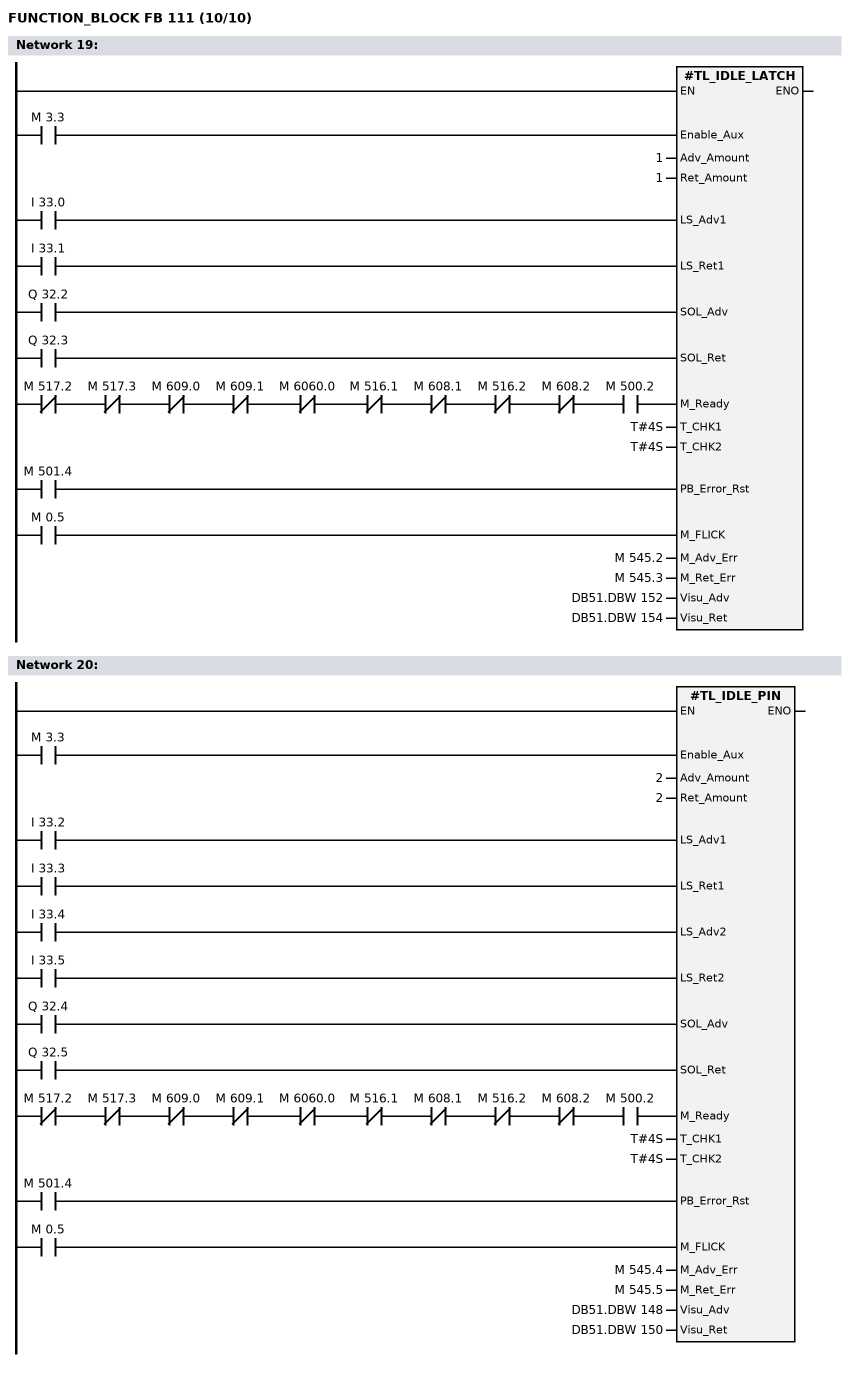

      A     M      3.3;
      =     L      0.0;
      BLD   103;
      A     I     33.0;
      =     L      0.1;
      BLD   103;
      A     I     33.1;
      =     L      0.2;
      BLD   103;
      A     Q     32.2;
      =     L      1.1;
      BLD   103;
      A     Q     32.3;
      =     L      1.2;
      BLD   103;
      AN    M    517.2;
      AN    M    517.3;
      AN    M    609.0;
      AN    M    609.1;
      AN    M   6060.0;
      AN    M    516.1;
      AN    M    608.1;
      AN    M    516.2;
      AN    M    608.2;
      A     M    500.2;
      =     L      1.3;
      BLD   103;
      A     M    501.4;
      =     L      1.5;
      BLD   103;
      A     M      0.5;
      =     L      1.6;
      BLD   103;
      CALL #TL_IDLE_LATCH (
           Enable_Aux               := L      0.0,
           Adv_Amount               := 1,
           Ret_Amount               := 1,
           LS_Adv1                  := L      0.1,
           LS_Ret1                  := L      0.2,
           SOL_Adv                  := L      1.1,
           SOL_Ret                  := L      1.2,
           M_Ready                  := L      1.3,
           T_CHK1                   := T#4S,
           T_CHK2                   := T#4S,
           PB_Error_Rst             := L      1.5,
           M_FLICK                  := L      1.6,
           M_Adv_Err                := M    545.2,
           M_Ret_Err                := M    545.3,
           Visu_Adv                 := DB51.DBW  152,
           Visu_Ret                 := DB51.DBW  154);
      NOP   0;
NETWORK
TITLE =

      A     M      3.3;
      =     L      0.0;
      BLD   103;
      A     I     33.2;
      =     L      0.1;
      BLD   103;
      A     I     33.3;
      =     L      0.2;
      BLD   103;
      A     I     33.4;
      =     L      0.3;
      BLD   103;
      A     I     33.5;
      =     L      0.4;
      BLD   103;
      A     Q     32.4;
      =     L      1.1;
      BLD   103;
      A     Q     32.5;
      =     L      1.2;
      BLD   103;
      AN    M    517.2;
      AN    M    517.3;
      AN    M    609.0;
      AN    M    609.1;
      AN    M   6060.0;
      AN    M    516.1;
      AN    M    608.1;
      AN    M    516.2;
      AN    M    608.2;
      A     M    500.2;
      =     L      1.3;
      BLD   103;
      A     M    501.4;
      =     L      1.5;
      BLD   103;
      A     M      0.5;
      =     L      1.6;
      BLD   103;
      CALL #TL_IDLE_PIN (
           Enable_Aux               := L      0.0,
           Adv_Amount               := 2,
           Ret_Amount               := 2,
           LS_Adv1                  := L      0.1,
           LS_Ret1                  := L      0.2,
           LS_Adv2                  := L      0.3,
           LS_Ret2                  := L      0.4,
           SOL_Adv                  := L      1.1,
           SOL_Ret                  := L      1.2,
           M_Ready                  := L      1.3,
           T_CHK1                   := T#4S,
           T_CHK2                   := T#4S,
           PB_Error_Rst             := L      1.5,
           M_FLICK                  := L      1.6,
           M_Adv_Err                := M    545.4,
           M_Ret_Err                := M    545.5,
           Visu_Adv                 := DB51.DBW  148,
           Visu_Ret                 := DB51.DBW  150);
      NOP   0;
END_FUNCTION_BLOCK

DATA_BLOCK DB 111
TITLE =
VERSION : 0.0

 FB 111
BEGIN
   LM_PIN.Enable_Aux := FALSE;
   LM_PIN.Adv_Amount := 0;
   LM_PIN.Ret_Amount := 0;
   LM_PIN.LS_Adv1 := FALSE;
   LM_PIN.LS_Ret1 := FALSE;
   LM_PIN.LS_Adv2 := FALSE;
   LM_PIN.LS_Ret2 := FALSE;
   LM_PIN.LS_Adv3 := FALSE;
   LM_PIN.LS_Ret3 := FALSE;
   LM_PIN.LS_Adv4 := FALSE;
   LM_PIN.LS_Ret4 := FALSE;
   LM_PIN.SOL_Adv := FALSE;
   LM_PIN.SOL_Ret := FALSE;
   LM_PIN.M_Ready := FALSE;
   LM_PIN.T_CHK1 := T#0MS;
   LM_PIN.T_CHK2 := T#0MS;
   LM_PIN.PB_Lamp_CHK := FALSE;
   LM_PIN.PB_Error_Rst := FALSE;
   LM_PIN.M_FLICK := FALSE;
   LM_PIN.M_Adv_Err := FALSE;
   LM_PIN.M_Ret_Err := FALSE;
   LM_PIN.LP_Adv := FALSE;
   LM_PIN.LP_Ret := FALSE;
   LM_PIN.Visu_Adv := W#16#0;
   LM_PIN.Visu_Ret := W#16#0;
   LM_PIN.Error_T1.IN := FALSE;
   LM_PIN.Error_T1.PT := T#0MS;
   LM_PIN.Error_T1.Q := FALSE;
   LM_PIN.Error_T1.ET := T#0MS;
   LM_PIN.Error_T1.STATE := B#16#0;
   LM_PIN.Error_T1.STIME := T#0MS;
   LM_PIN.Error_T1.ATIME := T#0MS;
   LM_PIN.Error_T2.IN := FALSE;
   LM_PIN.Error_T2.PT := T#0MS;
   LM_PIN.Error_T2.Q := FALSE;
   LM_PIN.Error_T2.ET := T#0MS;
   LM_PIN.Error_T2.STATE := B#16#0;
   LM_PIN.Error_T2.STIME := T#0MS;
   LM_PIN.Error_T2.ATIME := T#0MS;
   LM_PIN.CHK_Aux1 := FALSE;
   LM_PIN.CHK_Aux2 := FALSE;
   LM_PIN.Error_T1_DN := FALSE;
   LM_PIN.Error_T2_DN := FALSE;
   LM_PIN.Adv_Memo := FALSE;
   LM_PIN.Visu_Adv_Arr[0] := FALSE;
   LM_PIN.Visu_Adv_Arr[1] := FALSE;
   LM_PIN.Visu_Adv_Arr[2] := FALSE;
   LM_PIN.Visu_Adv_Arr[3] := FALSE;
   LM_PIN.Visu_Adv_Arr[4] := FALSE;
   LM_PIN.Visu_Adv_Arr[5] := FALSE;
   LM_PIN.Visu_Adv_Arr[6] := FALSE;
   LM_PIN.Visu_Adv_Arr[7] := FALSE;
   LM_PIN.Visu_Adv_Arr[8] := FALSE;
   LM_PIN.Visu_Adv_Arr[9] := FALSE;
   LM_PIN.Visu_Adv_Arr[10] := FALSE;
   LM_PIN.Visu_Adv_Arr[11] := FALSE;
   LM_PIN.Visu_Adv_Arr[12] := FALSE;
   LM_PIN.Visu_Adv_Arr[13] := FALSE;
   LM_PIN.Visu_Adv_Arr[14] := FALSE;
   LM_PIN.Visu_Adv_Arr[15] := FALSE;
   LM_PIN.Visu_Ret_Arr[0] := FALSE;
   LM_PIN.Visu_Ret_Arr[1] := FALSE;
   LM_PIN.Visu_Ret_Arr[2] := FALSE;
   LM_PIN.Visu_Ret_Arr[3] := FALSE;
   LM_PIN.Visu_Ret_Arr[4] := FALSE;
   LM_PIN.Visu_Ret_Arr[5] := FALSE;
   LM_PIN.Visu_Ret_Arr[6] := FALSE;
   LM_PIN.Visu_Ret_Arr[7] := FALSE;
   LM_PIN.Visu_Ret_Arr[8] := FALSE;
   LM_PIN.Visu_Ret_Arr[9] := FALSE;
   LM_PIN.Visu_Ret_Arr[10] := FALSE;
   LM_PIN.Visu_Ret_Arr[11] := FALSE;
   LM_PIN.Visu_Ret_Arr[12] := FALSE;
   LM_PIN.Visu_Ret_Arr[13] := FALSE;
   LM_PIN.Visu_Ret_Arr[14] := FALSE;
   LM_PIN.Visu_Ret_Arr[15] := FALSE;
   LM_PIN.BLK_Move_Ret := 0;
   LM_PIN.Enable := FALSE;
   LM_PIN.Adv_End := FALSE;
   LM_PIN.Ret_End := FALSE;
   LM_CLAMP1.Enable_Aux := FALSE;
   LM_CLAMP1.Adv_Amount := 0;
   LM_CLAMP1.Ret_Amount := 0;
   LM_CLAMP1.LS_Adv1 := FALSE;
   LM_CLAMP1.LS_Ret1 := FALSE;
   LM_CLAMP1.LS_Adv2 := FALSE;
   LM_CLAMP1.LS_Ret2 := FALSE;
   LM_CLAMP1.LS_Adv3 := FALSE;
   LM_CLAMP1.LS_Ret3 := FALSE;
   LM_CLAMP1.LS_Adv4 := FALSE;
   LM_CLAMP1.LS_Ret4 := FALSE;
   LM_CLAMP1.SOL_Adv := FALSE;
   LM_CLAMP1.SOL_Ret := FALSE;
   LM_CLAMP1.M_Ready := FALSE;
   LM_CLAMP1.T_CHK1 := T#0MS;
   LM_CLAMP1.T_CHK2 := T#0MS;
   LM_CLAMP1.PB_Lamp_CHK := FALSE;
   LM_CLAMP1.PB_Error_Rst := FALSE;
   LM_CLAMP1.M_FLICK := FALSE;
   LM_CLAMP1.M_Adv_Err := FALSE;
   LM_CLAMP1.M_Ret_Err := FALSE;
   LM_CLAMP1.LP_Adv := FALSE;
   LM_CLAMP1.LP_Ret := FALSE;
   LM_CLAMP1.Visu_Adv := W#16#0;
   LM_CLAMP1.Visu_Ret := W#16#0;
   LM_CLAMP1.Error_T1.IN := FALSE;
   LM_CLAMP1.Error_T1.PT := T#0MS;
   LM_CLAMP1.Error_T1.Q := FALSE;
   LM_CLAMP1.Error_T1.ET := T#0MS;
   LM_CLAMP1.Error_T1.STATE := B#16#0;
   LM_CLAMP1.Error_T1.STIME := T#0MS;
   LM_CLAMP1.Error_T1.ATIME := T#0MS;
   LM_CLAMP1.Error_T2.IN := FALSE;
   LM_CLAMP1.Error_T2.PT := T#0MS;
   LM_CLAMP1.Error_T2.Q := FALSE;
   LM_CLAMP1.Error_T2.ET := T#0MS;
   LM_CLAMP1.Error_T2.STATE := B#16#0;
   LM_CLAMP1.Error_T2.STIME := T#0MS;
   LM_CLAMP1.Error_T2.ATIME := T#0MS;
   LM_CLAMP1.CHK_Aux1 := FALSE;
   LM_CLAMP1.CHK_Aux2 := FALSE;
   LM_CLAMP1.Error_T1_DN := FALSE;
   LM_CLAMP1.Error_T2_DN := FALSE;
   LM_CLAMP1.Adv_Memo := FALSE;
   LM_CLAMP1.Visu_Adv_Arr[0] := FALSE;
   LM_CLAMP1.Visu_Adv_Arr[1] := FALSE;
   LM_CLAMP1.Visu_Adv_Arr[2] := FALSE;
   LM_CLAMP1.Visu_Adv_Arr[3] := FALSE;
   LM_CLAMP1.Visu_Adv_Arr[4] := FALSE;
   LM_CLAMP1.Visu_Adv_Arr[5] := FALSE;
   LM_CLAMP1.Visu_Adv_Arr[6] := FALSE;
   LM_CLAMP1.Visu_Adv_Arr[7] := FALSE;
   LM_CLAMP1.Visu_Adv_Arr[8] := FALSE;
   LM_CLAMP1.Visu_Adv_Arr[9] := FALSE;
   LM_CLAMP1.Visu_Adv_Arr[10] := FALSE;
   LM_CLAMP1.Visu_Adv_Arr[11] := FALSE;
   LM_CLAMP1.Visu_Adv_Arr[12] := FALSE;
   LM_CLAMP1.Visu_Adv_Arr[13] := FALSE;
   LM_CLAMP1.Visu_Adv_Arr[14] := FALSE;
   LM_CLAMP1.Visu_Adv_Arr[15] := FALSE;
   LM_CLAMP1.Visu_Ret_Arr[0] := FALSE;
   LM_CLAMP1.Visu_Ret_Arr[1] := FALSE;
   LM_CLAMP1.Visu_Ret_Arr[2] := FALSE;
   LM_CLAMP1.Visu_Ret_Arr[3] := FALSE;
   LM_CLAMP1.Visu_Ret_Arr[4] := FALSE;
   LM_CLAMP1.Visu_Ret_Arr[5] := FALSE;
   LM_CLAMP1.Visu_Ret_Arr[6] := FALSE;
   LM_CLAMP1.Visu_Ret_Arr[7] := FALSE;
   LM_CLAMP1.Visu_Ret_Arr[8] := FALSE;
   LM_CLAMP1.Visu_Ret_Arr[9] := FALSE;
   LM_CLAMP1.Visu_Ret_Arr[10] := FALSE;
   LM_CLAMP1.Visu_Ret_Arr[11] := FALSE;
   LM_CLAMP1.Visu_Ret_Arr[12] := FALSE;
   LM_CLAMP1.Visu_Ret_Arr[13] := FALSE;
   LM_CLAMP1.Visu_Ret_Arr[14] := FALSE;
   LM_CLAMP1.Visu_Ret_Arr[15] := FALSE;
   LM_CLAMP1.BLK_Move_Ret := 0;
   LM_CLAMP1.Enable := FALSE;
   LM_CLAMP1.Adv_End := FALSE;
   LM_CLAMP1.Ret_End := FALSE;
   LM_CLAMP2.Enable_Aux := FALSE;
   LM_CLAMP2.Adv_Amount := 0;
   LM_CLAMP2.Ret_Amount := 0;
   LM_CLAMP2.LS_Adv1 := FALSE;
   LM_CLAMP2.LS_Ret1 := FALSE;
   LM_CLAMP2.LS_Adv2 := FALSE;
   LM_CLAMP2.LS_Ret2 := FALSE;
   LM_CLAMP2.LS_Adv3 := FALSE;
   LM_CLAMP2.LS_Ret3 := FALSE;
   LM_CLAMP2.LS_Adv4 := FALSE;
   LM_CLAMP2.LS_Ret4 := FALSE;
   LM_CLAMP2.SOL_Adv := FALSE;
   LM_CLAMP2.SOL_Ret := FALSE;
   LM_CLAMP2.M_Ready := FALSE;
   LM_CLAMP2.T_CHK1 := T#0MS;
   LM_CLAMP2.T_CHK2 := T#0MS;
   LM_CLAMP2.PB_Lamp_CHK := FALSE;
   LM_CLAMP2.PB_Error_Rst := FALSE;
   LM_CLAMP2.M_FLICK := FALSE;
   LM_CLAMP2.M_Adv_Err := FALSE;
   LM_CLAMP2.M_Ret_Err := FALSE;
   LM_CLAMP2.LP_Adv := FALSE;
   LM_CLAMP2.LP_Ret := FALSE;
   LM_CLAMP2.Visu_Adv := W#16#0;
   LM_CLAMP2.Visu_Ret := W#16#0;
   LM_CLAMP2.Error_T1.IN := FALSE;
   LM_CLAMP2.Error_T1.PT := T#0MS;
   LM_CLAMP2.Error_T1.Q := FALSE;
   LM_CLAMP2.Error_T1.ET := T#0MS;
   LM_CLAMP2.Error_T1.STATE := B#16#0;
   LM_CLAMP2.Error_T1.STIME := T#0MS;
   LM_CLAMP2.Error_T1.ATIME := T#0MS;
   LM_CLAMP2.Error_T2.IN := FALSE;
   LM_CLAMP2.Error_T2.PT := T#0MS;
   LM_CLAMP2.Error_T2.Q := FALSE;
   LM_CLAMP2.Error_T2.ET := T#0MS;
   LM_CLAMP2.Error_T2.STATE := B#16#0;
   LM_CLAMP2.Error_T2.STIME := T#0MS;
   LM_CLAMP2.Error_T2.ATIME := T#0MS;
   LM_CLAMP2.CHK_Aux1 := FALSE;
   LM_CLAMP2.CHK_Aux2 := FALSE;
   LM_CLAMP2.Error_T1_DN := FALSE;
   LM_CLAMP2.Error_T2_DN := FALSE;
   LM_CLAMP2.Adv_Memo := FALSE;
   LM_CLAMP2.Visu_Adv_Arr[0] := FALSE;
   LM_CLAMP2.Visu_Adv_Arr[1] := FALSE;
   LM_CLAMP2.Visu_Adv_Arr[2] := FALSE;
   LM_CLAMP2.Visu_Adv_Arr[3] := FALSE;
   LM_CLAMP2.Visu_Adv_Arr[4] := FALSE;
   LM_CLAMP2.Visu_Adv_Arr[5] := FALSE;
   LM_CLAMP2.Visu_Adv_Arr[6] := FALSE;
   LM_CLAMP2.Visu_Adv_Arr[7] := FALSE;
   LM_CLAMP2.Visu_Adv_Arr[8] := FALSE;
   LM_CLAMP2.Visu_Adv_Arr[9] := FALSE;
   LM_CLAMP2.Visu_Adv_Arr[10] := FALSE;
   LM_CLAMP2.Visu_Adv_Arr[11] := FALSE;
   LM_CLAMP2.Visu_Adv_Arr[12] := FALSE;
   LM_CLAMP2.Visu_Adv_Arr[13] := FALSE;
   LM_CLAMP2.Visu_Adv_Arr[14] := FALSE;
   LM_CLAMP2.Visu_Adv_Arr[15] := FALSE;
   LM_CLAMP2.Visu_Ret_Arr[0] := FALSE;
   LM_CLAMP2.Visu_Ret_Arr[1] := FALSE;
   LM_CLAMP2.Visu_Ret_Arr[2] := FALSE;
   LM_CLAMP2.Visu_Ret_Arr[3] := FALSE;
   LM_CLAMP2.Visu_Ret_Arr[4] := FALSE;
   LM_CLAMP2.Visu_Ret_Arr[5] := FALSE;
   LM_CLAMP2.Visu_Ret_Arr[6] := FALSE;
   LM_CLAMP2.Visu_Ret_Arr[7] := FALSE;
   LM_CLAMP2.Visu_Ret_Arr[8] := FALSE;
   LM_CLAMP2.Visu_Ret_Arr[9] := FALSE;
   LM_CLAMP2.Visu_Ret_Arr[10] := FALSE;
   LM_CLAMP2.Visu_Ret_Arr[11] := FALSE;
   LM_CLAMP2.Visu_Ret_Arr[12] := FALSE;
   LM_CLAMP2.Visu_Ret_Arr[13] := FALSE;
   LM_CLAMP2.Visu_Ret_Arr[14] := FALSE;
   LM_CLAMP2.Visu_Ret_Arr[15] := FALSE;
   LM_CLAMP2.BLK_Move_Ret := 0;
   LM_CLAMP2.Enable := FALSE;
   LM_CLAMP2.Adv_End := FALSE;
   LM_CLAMP2.Ret_End := FALSE;
   LM_SLIDE.Enable_Aux := FALSE;
   LM_SLIDE.Adv_Amount := 0;
   LM_SLIDE.Ret_Amount := 0;
   LM_SLIDE.LS_Adv1 := FALSE;
   LM_SLIDE.LS_Ret1 := FALSE;
   LM_SLIDE.LS_Adv2 := FALSE;
   LM_SLIDE.LS_Ret2 := FALSE;
   LM_SLIDE.LS_Adv3 := FALSE;
   LM_SLIDE.LS_Ret3 := FALSE;
   LM_SLIDE.LS_Adv4 := FALSE;
   LM_SLIDE.LS_Ret4 := FALSE;
   LM_SLIDE.SOL_Adv := FALSE;
   LM_SLIDE.SOL_Ret := FALSE;
   LM_SLIDE.M_Ready := FALSE;
   LM_SLIDE.T_CHK1 := T#0MS;
   LM_SLIDE.T_CHK2 := T#0MS;
   LM_SLIDE.PB_Lamp_CHK := FALSE;
   LM_SLIDE.PB_Error_Rst := FALSE;
   LM_SLIDE.M_FLICK := FALSE;
   LM_SLIDE.M_Adv_Err := FALSE;
   LM_SLIDE.M_Ret_Err := FALSE;
   LM_SLIDE.LP_Adv := FALSE;
   LM_SLIDE.LP_Ret := FALSE;
   LM_SLIDE.Visu_Adv := W#16#0;
   LM_SLIDE.Visu_Ret := W#16#0;
   LM_SLIDE.Error_T1.IN := FALSE;
   LM_SLIDE.Error_T1.PT := T#0MS;
   LM_SLIDE.Error_T1.Q := FALSE;
   LM_SLIDE.Error_T1.ET := T#0MS;
   LM_SLIDE.Error_T1.STATE := B#16#0;
   LM_SLIDE.Error_T1.STIME := T#0MS;
   LM_SLIDE.Error_T1.ATIME := T#0MS;
   LM_SLIDE.Error_T2.IN := FALSE;
   LM_SLIDE.Error_T2.PT := T#0MS;
   LM_SLIDE.Error_T2.Q := FALSE;
   LM_SLIDE.Error_T2.ET := T#0MS;
   LM_SLIDE.Error_T2.STATE := B#16#0;
   LM_SLIDE.Error_T2.STIME := T#0MS;
   LM_SLIDE.Error_T2.ATIME := T#0MS;
   LM_SLIDE.CHK_Aux1 := FALSE;
   LM_SLIDE.CHK_Aux2 := FALSE;
   LM_SLIDE.Error_T1_DN := FALSE;
   LM_SLIDE.Error_T2_DN := FALSE;
   LM_SLIDE.Adv_Memo := FALSE;
   LM_SLIDE.Visu_Adv_Arr[0] := FALSE;
   LM_SLIDE.Visu_Adv_Arr[1] := FALSE;
   LM_SLIDE.Visu_Adv_Arr[2] := FALSE;
   LM_SLIDE.Visu_Adv_Arr[3] := FALSE;
   LM_SLIDE.Visu_Adv_Arr[4] := FALSE;
   LM_SLIDE.Visu_Adv_Arr[5] := FALSE;
   LM_SLIDE.Visu_Adv_Arr[6] := FALSE;
   LM_SLIDE.Visu_Adv_Arr[7] := FALSE;
   LM_SLIDE.Visu_Adv_Arr[8] := FALSE;
   LM_SLIDE.Visu_Adv_Arr[9] := FALSE;
   LM_SLIDE.Visu_Adv_Arr[10] := FALSE;
   LM_SLIDE.Visu_Adv_Arr[11] := FALSE;
   LM_SLIDE.Visu_Adv_Arr[12] := FALSE;
   LM_SLIDE.Visu_Adv_Arr[13] := FALSE;
   LM_SLIDE.Visu_Adv_Arr[14] := FALSE;
   LM_SLIDE.Visu_Adv_Arr[15] := FALSE;
   LM_SLIDE.Visu_Ret_Arr[0] := FALSE;
   LM_SLIDE.Visu_Ret_Arr[1] := FALSE;
   LM_SLIDE.Visu_Ret_Arr[2] := FALSE;
   LM_SLIDE.Visu_Ret_Arr[3] := FALSE;
   LM_SLIDE.Visu_Ret_Arr[4] := FALSE;
   LM_SLIDE.Visu_Ret_Arr[5] := FALSE;
   LM_SLIDE.Visu_Ret_Arr[6] := FALSE;
   LM_SLIDE.Visu_Ret_Arr[7] := FALSE;
   LM_SLIDE.Visu_Ret_Arr[8] := FALSE;
   LM_SLIDE.Visu_Ret_Arr[9] := FALSE;
   LM_SLIDE.Visu_Ret_Arr[10] := FALSE;
   LM_SLIDE.Visu_Ret_Arr[11] := FALSE;
   LM_SLIDE.Visu_Ret_Arr[12] := FALSE;
   LM_SLIDE.Visu_Ret_Arr[13] := FALSE;
   LM_SLIDE.Visu_Ret_Arr[14] := FALSE;
   LM_SLIDE.Visu_Ret_Arr[15] := FALSE;
   LM_SLIDE.BLK_Move_Ret := 0;
   LM_SLIDE.Enable := FALSE;
   LM_SLIDE.Adv_End := FALSE;
   LM_SLIDE.Ret_End := FALSE;
   LM_SLIDE_ADV_LOCK.Enable_Aux := FALSE;
   LM_SLIDE_ADV_LOCK.Adv_Amount := 0;
   LM_SLIDE_ADV_LOCK.Ret_Amount := 0;
   LM_SLIDE_ADV_LOCK.LS_Adv1 := FALSE;
   LM_SLIDE_ADV_LOCK.LS_Ret1 := FALSE;
   LM_SLIDE_ADV_LOCK.LS_Adv2 := FALSE;
   LM_SLIDE_ADV_LOCK.LS_Ret2 := FALSE;
   LM_SLIDE_ADV_LOCK.LS_Adv3 := FALSE;
   LM_SLIDE_ADV_LOCK.LS_Ret3 := FALSE;
   LM_SLIDE_ADV_LOCK.LS_Adv4 := FALSE;
   LM_SLIDE_ADV_LOCK.LS_Ret4 := FALSE;
   LM_SLIDE_ADV_LOCK.SOL_Adv := FALSE;
   LM_SLIDE_ADV_LOCK.SOL_Ret := FALSE;
   LM_SLIDE_ADV_LOCK.M_Ready := FALSE;
   LM_SLIDE_ADV_LOCK.T_CHK1 := T#0MS;
   LM_SLIDE_ADV_LOCK.T_CHK2 := T#0MS;
   LM_SLIDE_ADV_LOCK.PB_Lamp_CHK := FALSE;
   LM_SLIDE_ADV_LOCK.PB_Error_Rst := FALSE;
   LM_SLIDE_ADV_LOCK.M_FLICK := FALSE;
   LM_SLIDE_ADV_LOCK.M_Adv_Err := FALSE;
   LM_SLIDE_ADV_LOCK.M_Ret_Err := FALSE;
   LM_SLIDE_ADV_LOCK.LP_Adv := FALSE;
   LM_SLIDE_ADV_LOCK.LP_Ret := FALSE;
   LM_SLIDE_ADV_LOCK.Visu_Adv := W#16#0;
   LM_SLIDE_ADV_LOCK.Visu_Ret := W#16#0;
   LM_SLIDE_ADV_LOCK.Error_T1.IN := FALSE;
   LM_SLIDE_ADV_LOCK.Error_T1.PT := T#0MS;
   LM_SLIDE_ADV_LOCK.Error_T1.Q := FALSE;
   LM_SLIDE_ADV_LOCK.Error_T1.ET := T#0MS;
   LM_SLIDE_ADV_LOCK.Error_T1.STATE := B#16#0;
   LM_SLIDE_ADV_LOCK.Error_T1.STIME := T#0MS;
   LM_SLIDE_ADV_LOCK.Error_T1.ATIME := T#0MS;
   LM_SLIDE_ADV_LOCK.Error_T2.IN := FALSE;
   LM_SLIDE_ADV_LOCK.Error_T2.PT := T#0MS;
   LM_SLIDE_ADV_LOCK.Error_T2.Q := FALSE;
   LM_SLIDE_ADV_LOCK.Error_T2.ET := T#0MS;
   LM_SLIDE_ADV_LOCK.Error_T2.STATE := B#16#0;
   LM_SLIDE_ADV_LOCK.Error_T2.STIME := T#0MS;
   LM_SLIDE_ADV_LOCK.Error_T2.ATIME := T#0MS;
   LM_SLIDE_ADV_LOCK.CHK_Aux1 := FALSE;
   LM_SLIDE_ADV_LOCK.CHK_Aux2 := FALSE;
   LM_SLIDE_ADV_LOCK.Error_T1_DN := FALSE;
   LM_SLIDE_ADV_LOCK.Error_T2_DN := FALSE;
   LM_SLIDE_ADV_LOCK.Adv_Memo := FALSE;
   LM_SLIDE_ADV_LOCK.Visu_Adv_Arr[0] := FALSE;
   LM_SLIDE_ADV_LOCK.Visu_Adv_Arr[1] := FALSE;
   LM_SLIDE_ADV_LOCK.Visu_Adv_Arr[2] := FALSE;
   LM_SLIDE_ADV_LOCK.Visu_Adv_Arr[3] := FALSE;
   LM_SLIDE_ADV_LOCK.Visu_Adv_Arr[4] := FALSE;
   LM_SLIDE_ADV_LOCK.Visu_Adv_Arr[5] := FALSE;
   LM_SLIDE_ADV_LOCK.Visu_Adv_Arr[6] := FALSE;
   LM_SLIDE_ADV_LOCK.Visu_Adv_Arr[7] := FALSE;
   LM_SLIDE_ADV_LOCK.Visu_Adv_Arr[8] := FALSE;
   LM_SLIDE_ADV_LOCK.Visu_Adv_Arr[9] := FALSE;
   LM_SLIDE_ADV_LOCK.Visu_Adv_Arr[10] := FALSE;
   LM_SLIDE_ADV_LOCK.Visu_Adv_Arr[11] := FALSE;
   LM_SLIDE_ADV_LOCK.Visu_Adv_Arr[12] := FALSE;
   LM_SLIDE_ADV_LOCK.Visu_Adv_Arr[13] := FALSE;
   LM_SLIDE_ADV_LOCK.Visu_Adv_Arr[14] := FALSE;
   LM_SLIDE_ADV_LOCK.Visu_Adv_Arr[15] := FALSE;
   LM_SLIDE_ADV_LOCK.Visu_Ret_Arr[0] := FALSE;
   LM_SLIDE_ADV_LOCK.Visu_Ret_Arr[1] := FALSE;
   LM_SLIDE_ADV_LOCK.Visu_Ret_Arr[2] := FALSE;
   LM_SLIDE_ADV_LOCK.Visu_Ret_Arr[3] := FALSE;
   LM_SLIDE_ADV_LOCK.Visu_Ret_Arr[4] := FALSE;
   LM_SLIDE_ADV_LOCK.Visu_Ret_Arr[5] := FALSE;
   LM_SLIDE_ADV_LOCK.Visu_Ret_Arr[6] := FALSE;
   LM_SLIDE_ADV_LOCK.Visu_Ret_Arr[7] := FALSE;
   LM_SLIDE_ADV_LOCK.Visu_Ret_Arr[8] := FALSE;
   LM_SLIDE_ADV_LOCK.Visu_Ret_Arr[9] := FALSE;
   LM_SLIDE_ADV_LOCK.Visu_Ret_Arr[10] := FALSE;
   LM_SLIDE_ADV_LOCK.Visu_Ret_Arr[11] := FALSE;
   LM_SLIDE_ADV_LOCK.Visu_Ret_Arr[12] := FALSE;
   LM_SLIDE_ADV_LOCK.Visu_Ret_Arr[13] := FALSE;
   LM_SLIDE_ADV_LOCK.Visu_Ret_Arr[14] := FALSE;
   LM_SLIDE_ADV_LOCK.Visu_Ret_Arr[15] := FALSE;
   LM_SLIDE_ADV_LOCK.BLK_Move_Ret := 0;
   LM_SLIDE_ADV_LOCK.Enable := FALSE;
   LM_SLIDE_ADV_LOCK.Adv_End := FALSE;
   LM_SLIDE_ADV_LOCK.Ret_End := FALSE;
   LM_GUN1_SHIFT.Enable_Aux := FALSE;
   LM_GUN1_SHIFT.Adv_Amount := 0;
   LM_GUN1_SHIFT.Ret_Amount := 0;
   LM_GUN1_SHIFT.LS_Adv1 := FALSE;
   LM_GUN1_SHIFT.LS_Ret1 := FALSE;
   LM_GUN1_SHIFT.LS_Adv2 := FALSE;
   LM_GUN1_SHIFT.LS_Ret2 := FALSE;
   LM_GUN1_SHIFT.LS_Adv3 := FALSE;
   LM_GUN1_SHIFT.LS_Ret3 := FALSE;
   LM_GUN1_SHIFT.LS_Adv4 := FALSE;
   LM_GUN1_SHIFT.LS_Ret4 := FALSE;
   LM_GUN1_SHIFT.SOL_Adv := FALSE;
   LM_GUN1_SHIFT.SOL_Ret := FALSE;
   LM_GUN1_SHIFT.M_Ready := FALSE;
   LM_GUN1_SHIFT.T_CHK1 := T#0MS;
   LM_GUN1_SHIFT.T_CHK2 := T#0MS;
   LM_GUN1_SHIFT.PB_Lamp_CHK := FALSE;
   LM_GUN1_SHIFT.PB_Error_Rst := FALSE;
   LM_GUN1_SHIFT.M_FLICK := FALSE;
   LM_GUN1_SHIFT.M_Adv_Err := FALSE;
   LM_GUN1_SHIFT.M_Ret_Err := FALSE;
   LM_GUN1_SHIFT.LP_Adv := FALSE;
   LM_GUN1_SHIFT.LP_Ret := FALSE;
   LM_GUN1_SHIFT.Visu_Adv := W#16#0;
   LM_GUN1_SHIFT.Visu_Ret := W#16#0;
   LM_GUN1_SHIFT.Error_T1.IN := FALSE;
   LM_GUN1_SHIFT.Error_T1.PT := T#0MS;
   LM_GUN1_SHIFT.Error_T1.Q := FALSE;
   LM_GUN1_SHIFT.Error_T1.ET := T#0MS;
   LM_GUN1_SHIFT.Error_T1.STATE := B#16#0;
   LM_GUN1_SHIFT.Error_T1.STIME := T#0MS;
   LM_GUN1_SHIFT.Error_T1.ATIME := T#0MS;
   LM_GUN1_SHIFT.Error_T2.IN := FALSE;
   LM_GUN1_SHIFT.Error_T2.PT := T#0MS;
   LM_GUN1_SHIFT.Error_T2.Q := FALSE;
   LM_GUN1_SHIFT.Error_T2.ET := T#0MS;
   LM_GUN1_SHIFT.Error_T2.STATE := B#16#0;
   LM_GUN1_SHIFT.Error_T2.STIME := T#0MS;
   LM_GUN1_SHIFT.Error_T2.ATIME := T#0MS;
   LM_GUN1_SHIFT.CHK_Aux1 := FALSE;
   LM_GUN1_SHIFT.CHK_Aux2 := FALSE;
   LM_GUN1_SHIFT.Error_T1_DN := FALSE;
   LM_GUN1_SHIFT.Error_T2_DN := FALSE;
   LM_GUN1_SHIFT.Adv_Memo := FALSE;
   LM_GUN1_SHIFT.Visu_Adv_Arr[0] := FALSE;
   LM_GUN1_SHIFT.Visu_Adv_Arr[1] := FALSE;
   LM_GUN1_SHIFT.Visu_Adv_Arr[2] := FALSE;
   LM_GUN1_SHIFT.Visu_Adv_Arr[3] := FALSE;
   LM_GUN1_SHIFT.Visu_Adv_Arr[4] := FALSE;
   LM_GUN1_SHIFT.Visu_Adv_Arr[5] := FALSE;
   LM_GUN1_SHIFT.Visu_Adv_Arr[6] := FALSE;
   LM_GUN1_SHIFT.Visu_Adv_Arr[7] := FALSE;
   LM_GUN1_SHIFT.Visu_Adv_Arr[8] := FALSE;
   LM_GUN1_SHIFT.Visu_Adv_Arr[9] := FALSE;
   LM_GUN1_SHIFT.Visu_Adv_Arr[10] := FALSE;
   LM_GUN1_SHIFT.Visu_Adv_Arr[11] := FALSE;
   LM_GUN1_SHIFT.Visu_Adv_Arr[12] := FALSE;
   LM_GUN1_SHIFT.Visu_Adv_Arr[13] := FALSE;
   LM_GUN1_SHIFT.Visu_Adv_Arr[14] := FALSE;
   LM_GUN1_SHIFT.Visu_Adv_Arr[15] := FALSE;
   LM_GUN1_SHIFT.Visu_Ret_Arr[0] := FALSE;
   LM_GUN1_SHIFT.Visu_Ret_Arr[1] := FALSE;
   LM_GUN1_SHIFT.Visu_Ret_Arr[2] := FALSE;
   LM_GUN1_SHIFT.Visu_Ret_Arr[3] := FALSE;
   LM_GUN1_SHIFT.Visu_Ret_Arr[4] := FALSE;
   LM_GUN1_SHIFT.Visu_Ret_Arr[5] := FALSE;
   LM_GUN1_SHIFT.Visu_Ret_Arr[6] := FALSE;
   LM_GUN1_SHIFT.Visu_Ret_Arr[7] := FALSE;
   LM_GUN1_SHIFT.Visu_Ret_Arr[8] := FALSE;
   LM_GUN1_SHIFT.Visu_Ret_Arr[9] := FALSE;
   LM_GUN1_SHIFT.Visu_Ret_Arr[10] := FALSE;
   LM_GUN1_SHIFT.Visu_Ret_Arr[11] := FALSE;
   LM_GUN1_SHIFT.Visu_Ret_Arr[12] := FALSE;
   LM_GUN1_SHIFT.Visu_Ret_Arr[13] := FALSE;
   LM_GUN1_SHIFT.Visu_Ret_Arr[14] := FALSE;
   LM_GUN1_SHIFT.Visu_Ret_Arr[15] := FALSE;
   LM_GUN1_SHIFT.BLK_Move_Ret := 0;
   LM_GUN1_SHIFT.Enable := FALSE;
   LM_GUN1_SHIFT.Adv_End := FALSE;
   LM_GUN1_SHIFT.Ret_End := FALSE;
   LM_GUN2_SHIFT.Enable_Aux := FALSE;
   LM_GUN2_SHIFT.Adv_Amount := 0;
   LM_GUN2_SHIFT.Ret_Amount := 0;
   LM_GUN2_SHIFT.LS_Adv1 := FALSE;
   LM_GUN2_SHIFT.LS_Ret1 := FALSE;
   LM_GUN2_SHIFT.LS_Adv2 := FALSE;
   LM_GUN2_SHIFT.LS_Ret2 := FALSE;
   LM_GUN2_SHIFT.LS_Adv3 := FALSE;
   LM_GUN2_SHIFT.LS_Ret3 := FALSE;
   LM_GUN2_SHIFT.LS_Adv4 := FALSE;
   LM_GUN2_SHIFT.LS_Ret4 := FALSE;
   LM_GUN2_SHIFT.SOL_Adv := FALSE;
   LM_GUN2_SHIFT.SOL_Ret := FALSE;
   LM_GUN2_SHIFT.M_Ready := FALSE;
   LM_GUN2_SHIFT.T_CHK1 := T#0MS;
   LM_GUN2_SHIFT.T_CHK2 := T#0MS;
   LM_GUN2_SHIFT.PB_Lamp_CHK := FALSE;
   LM_GUN2_SHIFT.PB_Error_Rst := FALSE;
   LM_GUN2_SHIFT.M_FLICK := FALSE;
   LM_GUN2_SHIFT.M_Adv_Err := FALSE;
   LM_GUN2_SHIFT.M_Ret_Err := FALSE;
   LM_GUN2_SHIFT.LP_Adv := FALSE;
   LM_GUN2_SHIFT.LP_Ret := FALSE;
   LM_GUN2_SHIFT.Visu_Adv := W#16#0;
   LM_GUN2_SHIFT.Visu_Ret := W#16#0;
   LM_GUN2_SHIFT.Error_T1.IN := FALSE;
   LM_GUN2_SHIFT.Error_T1.PT := T#0MS;
   LM_GUN2_SHIFT.Error_T1.Q := FALSE;
   LM_GUN2_SHIFT.Error_T1.ET := T#0MS;
   LM_GUN2_SHIFT.Error_T1.STATE := B#16#0;
   LM_GUN2_SHIFT.Error_T1.STIME := T#0MS;
   LM_GUN2_SHIFT.Error_T1.ATIME := T#0MS;
   LM_GUN2_SHIFT.Error_T2.IN := FALSE;
   LM_GUN2_SHIFT.Error_T2.PT := T#0MS;
   LM_GUN2_SHIFT.Error_T2.Q := FALSE;
   LM_GUN2_SHIFT.Error_T2.ET := T#0MS;
   LM_GUN2_SHIFT.Error_T2.STATE := B#16#0;
   LM_GUN2_SHIFT.Error_T2.STIME := T#0MS;
   LM_GUN2_SHIFT.Error_T2.ATIME := T#0MS;
   LM_GUN2_SHIFT.CHK_Aux1 := FALSE;
   LM_GUN2_SHIFT.CHK_Aux2 := FALSE;
   LM_GUN2_SHIFT.Error_T1_DN := FALSE;
   LM_GUN2_SHIFT.Error_T2_DN := FALSE;
   LM_GUN2_SHIFT.Adv_Memo := FALSE;
   LM_GUN2_SHIFT.Visu_Adv_Arr[0] := FALSE;
   LM_GUN2_SHIFT.Visu_Adv_Arr[1] := FALSE;
   LM_GUN2_SHIFT.Visu_Adv_Arr[2] := FALSE;
   LM_GUN2_SHIFT.Visu_Adv_Arr[3] := FALSE;
   LM_GUN2_SHIFT.Visu_Adv_Arr[4] := FALSE;
   LM_GUN2_SHIFT.Visu_Adv_Arr[5] := FALSE;
   LM_GUN2_SHIFT.Visu_Adv_Arr[6] := FALSE;
   LM_GUN2_SHIFT.Visu_Adv_Arr[7] := FALSE;
   LM_GUN2_SHIFT.Visu_Adv_Arr[8] := FALSE;
   LM_GUN2_SHIFT.Visu_Adv_Arr[9] := FALSE;
   LM_GUN2_SHIFT.Visu_Adv_Arr[10] := FALSE;
   LM_GUN2_SHIFT.Visu_Adv_Arr[11] := FALSE;
   LM_GUN2_SHIFT.Visu_Adv_Arr[12] := FALSE;
   LM_GUN2_SHIFT.Visu_Adv_Arr[13] := FALSE;
   LM_GUN2_SHIFT.Visu_Adv_Arr[14] := FALSE;
   LM_GUN2_SHIFT.Visu_Adv_Arr[15] := FALSE;
   LM_GUN2_SHIFT.Visu_Ret_Arr[0] := FALSE;
   LM_GUN2_SHIFT.Visu_Ret_Arr[1] := FALSE;
   LM_GUN2_SHIFT.Visu_Ret_Arr[2] := FALSE;
   LM_GUN2_SHIFT.Visu_Ret_Arr[3] := FALSE;
   LM_GUN2_SHIFT.Visu_Ret_Arr[4] := FALSE;
   LM_GUN2_SHIFT.Visu_Ret_Arr[5] := FALSE;
   LM_GUN2_SHIFT.Visu_Ret_Arr[6] := FALSE;
   LM_GUN2_SHIFT.Visu_Ret_Arr[7] := FALSE;
   LM_GUN2_SHIFT.Visu_Ret_Arr[8] := FALSE;
   LM_GUN2_SHIFT.Visu_Ret_Arr[9] := FALSE;
   LM_GUN2_SHIFT.Visu_Ret_Arr[10] := FALSE;
   LM_GUN2_SHIFT.Visu_Ret_Arr[11] := FALSE;
   LM_GUN2_SHIFT.Visu_Ret_Arr[12] := FALSE;
   LM_GUN2_SHIFT.Visu_Ret_Arr[13] := FALSE;
   LM_GUN2_SHIFT.Visu_Ret_Arr[14] := FALSE;
   LM_GUN2_SHIFT.Visu_Ret_Arr[15] := FALSE;
   LM_GUN2_SHIFT.BLK_Move_Ret := 0;
   LM_GUN2_SHIFT.Enable := FALSE;
   LM_GUN2_SHIFT.Adv_End := FALSE;
   LM_GUN2_SHIFT.Ret_End := FALSE;
   LM_GUN2_LATCH.Enable_Aux := FALSE;
   LM_GUN2_LATCH.Adv_Amount := 0;
   LM_GUN2_LATCH.Ret_Amount := 0;
   LM_GUN2_LATCH.LS_Adv1 := FALSE;
   LM_GUN2_LATCH.LS_Ret1 := FALSE;
   LM_GUN2_LATCH.LS_Adv2 := FALSE;
   LM_GUN2_LATCH.LS_Ret2 := FALSE;
   LM_GUN2_LATCH.LS_Adv3 := FALSE;
   LM_GUN2_LATCH.LS_Ret3 := FALSE;
   LM_GUN2_LATCH.LS_Adv4 := FALSE;
   LM_GUN2_LATCH.LS_Ret4 := FALSE;
   LM_GUN2_LATCH.SOL_Adv := FALSE;
   LM_GUN2_LATCH.SOL_Ret := FALSE;
   LM_GUN2_LATCH.M_Ready := FALSE;
   LM_GUN2_LATCH.T_CHK1 := T#0MS;
   LM_GUN2_LATCH.T_CHK2 := T#0MS;
   LM_GUN2_LATCH.PB_Lamp_CHK := FALSE;
   LM_GUN2_LATCH.PB_Error_Rst := FALSE;
   LM_GUN2_LATCH.M_FLICK := FALSE;
   LM_GUN2_LATCH.M_Adv_Err := FALSE;
   LM_GUN2_LATCH.M_Ret_Err := FALSE;
   LM_GUN2_LATCH.LP_Adv := FALSE;
   LM_GUN2_LATCH.LP_Ret := FALSE;
   LM_GUN2_LATCH.Visu_Adv := W#16#0;
   LM_GUN2_LATCH.Visu_Ret := W#16#0;
   LM_GUN2_LATCH.Error_T1.IN := FALSE;
   LM_GUN2_LATCH.Error_T1.PT := T#0MS;
   LM_GUN2_LATCH.Error_T1.Q := FALSE;
   LM_GUN2_LATCH.Error_T1.ET := T#0MS;
   LM_GUN2_LATCH.Error_T1.STATE := B#16#0;
   LM_GUN2_LATCH.Error_T1.STIME := T#0MS;
   LM_GUN2_LATCH.Error_T1.ATIME := T#0MS;
   LM_GUN2_LATCH.Error_T2.IN := FALSE;
   LM_GUN2_LATCH.Error_T2.PT := T#0MS;
   LM_GUN2_LATCH.Error_T2.Q := FALSE;
   LM_GUN2_LATCH.Error_T2.ET := T#0MS;
   LM_GUN2_LATCH.Error_T2.STATE := B#16#0;
   LM_GUN2_LATCH.Error_T2.STIME := T#0MS;
   LM_GUN2_LATCH.Error_T2.ATIME := T#0MS;
   LM_GUN2_LATCH.CHK_Aux1 := FALSE;
   LM_GUN2_LATCH.CHK_Aux2 := FALSE;
   LM_GUN2_LATCH.Error_T1_DN := FALSE;
   LM_GUN2_LATCH.Error_T2_DN := FALSE;
   LM_GUN2_LATCH.Adv_Memo := FALSE;
   LM_GUN2_LATCH.Visu_Adv_Arr[0] := FALSE;
   LM_GUN2_LATCH.Visu_Adv_Arr[1] := FALSE;
   LM_GUN2_LATCH.Visu_Adv_Arr[2] := FALSE;
   LM_GUN2_LATCH.Visu_Adv_Arr[3] := FALSE;
   LM_GUN2_LATCH.Visu_Adv_Arr[4] := FALSE;
   LM_GUN2_LATCH.Visu_Adv_Arr[5] := FALSE;
   LM_GUN2_LATCH.Visu_Adv_Arr[6] := FALSE;
   LM_GUN2_LATCH.Visu_Adv_Arr[7] := FALSE;
   LM_GUN2_LATCH.Visu_Adv_Arr[8] := FALSE;
   LM_GUN2_LATCH.Visu_Adv_Arr[9] := FALSE;
   LM_GUN2_LATCH.Visu_Adv_Arr[10] := FALSE;
   LM_GUN2_LATCH.Visu_Adv_Arr[11] := FALSE;
   LM_GUN2_LATCH.Visu_Adv_Arr[12] := FALSE;
   LM_GUN2_LATCH.Visu_Adv_Arr[13] := FALSE;
   LM_GUN2_LATCH.Visu_Adv_Arr[14] := FALSE;
   LM_GUN2_LATCH.Visu_Adv_Arr[15] := FALSE;
   LM_GUN2_LATCH.Visu_Ret_Arr[0] := FALSE;
   LM_GUN2_LATCH.Visu_Ret_Arr[1] := FALSE;
   LM_GUN2_LATCH.Visu_Ret_Arr[2] := FALSE;
   LM_GUN2_LATCH.Visu_Ret_Arr[3] := FALSE;
   LM_GUN2_LATCH.Visu_Ret_Arr[4] := FALSE;
   LM_GUN2_LATCH.Visu_Ret_Arr[5] := FALSE;
   LM_GUN2_LATCH.Visu_Ret_Arr[6] := FALSE;
   LM_GUN2_LATCH.Visu_Ret_Arr[7] := FALSE;
   LM_GUN2_LATCH.Visu_Ret_Arr[8] := FALSE;
   LM_GUN2_LATCH.Visu_Ret_Arr[9] := FALSE;
   LM_GUN2_LATCH.Visu_Ret_Arr[10] := FALSE;
   LM_GUN2_LATCH.Visu_Ret_Arr[11] := FALSE;
   LM_GUN2_LATCH.Visu_Ret_Arr[12] := FALSE;
   LM_GUN2_LATCH.Visu_Ret_Arr[13] := FALSE;
   LM_GUN2_LATCH.Visu_Ret_Arr[14] := FALSE;
   LM_GUN2_LATCH.Visu_Ret_Arr[15] := FALSE;
   LM_GUN2_LATCH.BLK_Move_Ret := 0;
   LM_GUN2_LATCH.Enable := FALSE;
   LM_GUN2_LATCH.Adv_End := FALSE;
   LM_GUN2_LATCH.Ret_End := FALSE;
   TL_SLIDE.Enable_Aux := FALSE;
   TL_SLIDE.Adv_Amount := 0;
   TL_SLIDE.Ret_Amount := 0;
   TL_SLIDE.LS_Adv1 := FALSE;
   TL_SLIDE.LS_Ret1 := FALSE;
   TL_SLIDE.LS_Adv2 := FALSE;
   TL_SLIDE.LS_Ret2 := FALSE;
   TL_SLIDE.LS_Adv3 := FALSE;
   TL_SLIDE.LS_Ret3 := FALSE;
   TL_SLIDE.LS_Adv4 := FALSE;
   TL_SLIDE.LS_Ret4 := FALSE;
   TL_SLIDE.SOL_Adv := FALSE;
   TL_SLIDE.SOL_Ret := FALSE;
   TL_SLIDE.M_Ready := FALSE;
   TL_SLIDE.T_CHK1 := T#0MS;
   TL_SLIDE.T_CHK2 := T#0MS;
   TL_SLIDE.PB_Lamp_CHK := FALSE;
   TL_SLIDE.PB_Error_Rst := FALSE;
   TL_SLIDE.M_FLICK := FALSE;
   TL_SLIDE.M_Adv_Err := FALSE;
   TL_SLIDE.M_Ret_Err := FALSE;
   TL_SLIDE.LP_Adv := FALSE;
   TL_SLIDE.LP_Ret := FALSE;
   TL_SLIDE.Visu_Adv := W#16#0;
   TL_SLIDE.Visu_Ret := W#16#0;
   TL_SLIDE.Error_T1.IN := FALSE;
   TL_SLIDE.Error_T1.PT := T#0MS;
   TL_SLIDE.Error_T1.Q := FALSE;
   TL_SLIDE.Error_T1.ET := T#0MS;
   TL_SLIDE.Error_T1.STATE := B#16#0;
   TL_SLIDE.Error_T1.STIME := T#0MS;
   TL_SLIDE.Error_T1.ATIME := T#0MS;
   TL_SLIDE.Error_T2.IN := FALSE;
   TL_SLIDE.Error_T2.PT := T#0MS;
   TL_SLIDE.Error_T2.Q := FALSE;
   TL_SLIDE.Error_T2.ET := T#0MS;
   TL_SLIDE.Error_T2.STATE := B#16#0;
   TL_SLIDE.Error_T2.STIME := T#0MS;
   TL_SLIDE.Error_T2.ATIME := T#0MS;
   TL_SLIDE.CHK_Aux1 := FALSE;
   TL_SLIDE.CHK_Aux2 := FALSE;
   TL_SLIDE.Error_T1_DN := FALSE;
   TL_SLIDE.Error_T2_DN := FALSE;
   TL_SLIDE.Adv_Memo := FALSE;
   TL_SLIDE.Visu_Adv_Arr[0] := FALSE;
   TL_SLIDE.Visu_Adv_Arr[1] := FALSE;
   TL_SLIDE.Visu_Adv_Arr[2] := FALSE;
   TL_SLIDE.Visu_Adv_Arr[3] := FALSE;
   TL_SLIDE.Visu_Adv_Arr[4] := FALSE;
   TL_SLIDE.Visu_Adv_Arr[5] := FALSE;
   TL_SLIDE.Visu_Adv_Arr[6] := FALSE;
   TL_SLIDE.Visu_Adv_Arr[7] := FALSE;
   TL_SLIDE.Visu_Adv_Arr[8] := FALSE;
   TL_SLIDE.Visu_Adv_Arr[9] := FALSE;
   TL_SLIDE.Visu_Adv_Arr[10] := FALSE;
   TL_SLIDE.Visu_Adv_Arr[11] := FALSE;
   TL_SLIDE.Visu_Adv_Arr[12] := FALSE;
   TL_SLIDE.Visu_Adv_Arr[13] := FALSE;
   TL_SLIDE.Visu_Adv_Arr[14] := FALSE;
   TL_SLIDE.Visu_Adv_Arr[15] := FALSE;
   TL_SLIDE.Visu_Ret_Arr[0] := FALSE;
   TL_SLIDE.Visu_Ret_Arr[1] := FALSE;
   TL_SLIDE.Visu_Ret_Arr[2] := FALSE;
   TL_SLIDE.Visu_Ret_Arr[3] := FALSE;
   TL_SLIDE.Visu_Ret_Arr[4] := FALSE;
   TL_SLIDE.Visu_Ret_Arr[5] := FALSE;
   TL_SLIDE.Visu_Ret_Arr[6] := FALSE;
   TL_SLIDE.Visu_Ret_Arr[7] := FALSE;
   TL_SLIDE.Visu_Ret_Arr[8] := FALSE;
   TL_SLIDE.Visu_Ret_Arr[9] := FALSE;
   TL_SLIDE.Visu_Ret_Arr[10] := FALSE;
   TL_SLIDE.Visu_Ret_Arr[11] := FALSE;
   TL_SLIDE.Visu_Ret_Arr[12] := FALSE;
   TL_SLIDE.Visu_Ret_Arr[13] := FALSE;
   TL_SLIDE.Visu_Ret_Arr[14] := FALSE;
   TL_SLIDE.Visu_Ret_Arr[15] := FALSE;
   TL_SLIDE.BLK_Move_Ret := 0;
   TL_SLIDE.Enable := FALSE;
   TL_SLIDE.Adv_End := FALSE;
   TL_SLIDE.Ret_End := FALSE;
   TL_SLIDE_LOCK.Enable_Aux := FALSE;
   TL_SLIDE_LOCK.Adv_Amount := 0;
   TL_SLIDE_LOCK.Ret_Amount := 0;
   TL_SLIDE_LOCK.LS_Adv1 := FALSE;
   TL_SLIDE_LOCK.LS_Ret1 := FALSE;
   TL_SLIDE_LOCK.LS_Adv2 := FALSE;
   TL_SLIDE_LOCK.LS_Ret2 := FALSE;
   TL_SLIDE_LOCK.LS_Adv3 := FALSE;
   TL_SLIDE_LOCK.LS_Ret3 := FALSE;
   TL_SLIDE_LOCK.LS_Adv4 := FALSE;
   TL_SLIDE_LOCK.LS_Ret4 := FALSE;
   TL_SLIDE_LOCK.SOL_Adv := FALSE;
   TL_SLIDE_LOCK.SOL_Ret := FALSE;
   TL_SLIDE_LOCK.M_Ready := FALSE;
   TL_SLIDE_LOCK.T_CHK1 := T#0MS;
   TL_SLIDE_LOCK.T_CHK2 := T#0MS;
   TL_SLIDE_LOCK.PB_Lamp_CHK := FALSE;
   TL_SLIDE_LOCK.PB_Error_Rst := FALSE;
   TL_SLIDE_LOCK.M_FLICK := FALSE;
   TL_SLIDE_LOCK.M_Adv_Err := FALSE;
   TL_SLIDE_LOCK.M_Ret_Err := FALSE;
   TL_SLIDE_LOCK.LP_Adv := FALSE;
   TL_SLIDE_LOCK.LP_Ret := FALSE;
   TL_SLIDE_LOCK.Visu_Adv := W#16#0;
   TL_SLIDE_LOCK.Visu_Ret := W#16#0;
   TL_SLIDE_LOCK.Error_T1.IN := FALSE;
   TL_SLIDE_LOCK.Error_T1.PT := T#0MS;
   TL_SLIDE_LOCK.Error_T1.Q := FALSE;
   TL_SLIDE_LOCK.Error_T1.ET := T#0MS;
   TL_SLIDE_LOCK.Error_T1.STATE := B#16#0;
   TL_SLIDE_LOCK.Error_T1.STIME := T#0MS;
   TL_SLIDE_LOCK.Error_T1.ATIME := T#0MS;
   TL_SLIDE_LOCK.Error_T2.IN := FALSE;
   TL_SLIDE_LOCK.Error_T2.PT := T#0MS;
   TL_SLIDE_LOCK.Error_T2.Q := FALSE;
   TL_SLIDE_LOCK.Error_T2.ET := T#0MS;
   TL_SLIDE_LOCK.Error_T2.STATE := B#16#0;
   TL_SLIDE_LOCK.Error_T2.STIME := T#0MS;
   TL_SLIDE_LOCK.Error_T2.ATIME := T#0MS;
   TL_SLIDE_LOCK.CHK_Aux1 := FALSE;
   TL_SLIDE_LOCK.CHK_Aux2 := FALSE;
   TL_SLIDE_LOCK.Error_T1_DN := FALSE;
   TL_SLIDE_LOCK.Error_T2_DN := FALSE;
   TL_SLIDE_LOCK.Adv_Memo := FALSE;
   TL_SLIDE_LOCK.Visu_Adv_Arr[0] := FALSE;
   TL_SLIDE_LOCK.Visu_Adv_Arr[1] := FALSE;
   TL_SLIDE_LOCK.Visu_Adv_Arr[2] := FALSE;
   TL_SLIDE_LOCK.Visu_Adv_Arr[3] := FALSE;
   TL_SLIDE_LOCK.Visu_Adv_Arr[4] := FALSE;
   TL_SLIDE_LOCK.Visu_Adv_Arr[5] := FALSE;
   TL_SLIDE_LOCK.Visu_Adv_Arr[6] := FALSE;
   TL_SLIDE_LOCK.Visu_Adv_Arr[7] := FALSE;
   TL_SLIDE_LOCK.Visu_Adv_Arr[8] := FALSE;
   TL_SLIDE_LOCK.Visu_Adv_Arr[9] := FALSE;
   TL_SLIDE_LOCK.Visu_Adv_Arr[10] := FALSE;
   TL_SLIDE_LOCK.Visu_Adv_Arr[11] := FALSE;
   TL_SLIDE_LOCK.Visu_Adv_Arr[12] := FALSE;
   TL_SLIDE_LOCK.Visu_Adv_Arr[13] := FALSE;
   TL_SLIDE_LOCK.Visu_Adv_Arr[14] := FALSE;
   TL_SLIDE_LOCK.Visu_Adv_Arr[15] := FALSE;
   TL_SLIDE_LOCK.Visu_Ret_Arr[0] := FALSE;
   TL_SLIDE_LOCK.Visu_Ret_Arr[1] := FALSE;
   TL_SLIDE_LOCK.Visu_Ret_Arr[2] := FALSE;
   TL_SLIDE_LOCK.Visu_Ret_Arr[3] := FALSE;
   TL_SLIDE_LOCK.Visu_Ret_Arr[4] := FALSE;
   TL_SLIDE_LOCK.Visu_Ret_Arr[5] := FALSE;
   TL_SLIDE_LOCK.Visu_Ret_Arr[6] := FALSE;
   TL_SLIDE_LOCK.Visu_Ret_Arr[7] := FALSE;
   TL_SLIDE_LOCK.Visu_Ret_Arr[8] := FALSE;
   TL_SLIDE_LOCK.Visu_Ret_Arr[9] := FALSE;
   TL_SLIDE_LOCK.Visu_Ret_Arr[10] := FALSE;
   TL_SLIDE_LOCK.Visu_Ret_Arr[11] := FALSE;
   TL_SLIDE_LOCK.Visu_Ret_Arr[12] := FALSE;
   TL_SLIDE_LOCK.Visu_Ret_Arr[13] := FALSE;
   TL_SLIDE_LOCK.Visu_Ret_Arr[14] := FALSE;
   TL_SLIDE_LOCK.Visu_Ret_Arr[15] := FALSE;
   TL_SLIDE_LOCK.BLK_Move_Ret := 0;
   TL_SLIDE_LOCK.Enable := FALSE;
   TL_SLIDE_LOCK.Adv_End := FALSE;
   TL_SLIDE_LOCK.Ret_End := FALSE;
   TL_PIN_UP_DOWN.Enable_Aux := FALSE;
   TL_PIN_UP_DOWN.Adv_Amount := 0;
   TL_PIN_UP_DOWN.Ret_Amount := 0;
   TL_PIN_UP_DOWN.LS_Adv1 := FALSE;
   TL_PIN_UP_DOWN.LS_Ret1 := FALSE;
   TL_PIN_UP_DOWN.LS_Adv2 := FALSE;
   TL_PIN_UP_DOWN.LS_Ret2 := FALSE;
   TL_PIN_UP_DOWN.LS_Adv3 := FALSE;
   TL_PIN_UP_DOWN.LS_Ret3 := FALSE;
   TL_PIN_UP_DOWN.LS_Adv4 := FALSE;
   TL_PIN_UP_DOWN.LS_Ret4 := FALSE;
   TL_PIN_UP_DOWN.SOL_Adv := FALSE;
   TL_PIN_UP_DOWN.SOL_Ret := FALSE;
   TL_PIN_UP_DOWN.M_Ready := FALSE;
   TL_PIN_UP_DOWN.T_CHK1 := T#0MS;
   TL_PIN_UP_DOWN.T_CHK2 := T#0MS;
   TL_PIN_UP_DOWN.PB_Lamp_CHK := FALSE;
   TL_PIN_UP_DOWN.PB_Error_Rst := FALSE;
   TL_PIN_UP_DOWN.M_FLICK := FALSE;
   TL_PIN_UP_DOWN.M_Adv_Err := FALSE;
   TL_PIN_UP_DOWN.M_Ret_Err := FALSE;
   TL_PIN_UP_DOWN.LP_Adv := FALSE;
   TL_PIN_UP_DOWN.LP_Ret := FALSE;
   TL_PIN_UP_DOWN.Visu_Adv := W#16#0;
   TL_PIN_UP_DOWN.Visu_Ret := W#16#0;
   TL_PIN_UP_DOWN.Error_T1.IN := FALSE;
   TL_PIN_UP_DOWN.Error_T1.PT := T#0MS;
   TL_PIN_UP_DOWN.Error_T1.Q := FALSE;
   TL_PIN_UP_DOWN.Error_T1.ET := T#0MS;
   TL_PIN_UP_DOWN.Error_T1.STATE := B#16#0;
   TL_PIN_UP_DOWN.Error_T1.STIME := T#0MS;
   TL_PIN_UP_DOWN.Error_T1.ATIME := T#0MS;
   TL_PIN_UP_DOWN.Error_T2.IN := FALSE;
   TL_PIN_UP_DOWN.Error_T2.PT := T#0MS;
   TL_PIN_UP_DOWN.Error_T2.Q := FALSE;
   TL_PIN_UP_DOWN.Error_T2.ET := T#0MS;
   TL_PIN_UP_DOWN.Error_T2.STATE := B#16#0;
   TL_PIN_UP_DOWN.Error_T2.STIME := T#0MS;
   TL_PIN_UP_DOWN.Error_T2.ATIME := T#0MS;
   TL_PIN_UP_DOWN.CHK_Aux1 := FALSE;
   TL_PIN_UP_DOWN.CHK_Aux2 := FALSE;
   TL_PIN_UP_DOWN.Error_T1_DN := FALSE;
   TL_PIN_UP_DOWN.Error_T2_DN := FALSE;
   TL_PIN_UP_DOWN.Adv_Memo := FALSE;
   TL_PIN_UP_DOWN.Visu_Adv_Arr[0] := FALSE;
   TL_PIN_UP_DOWN.Visu_Adv_Arr[1] := FALSE;
   TL_PIN_UP_DOWN.Visu_Adv_Arr[2] := FALSE;
   TL_PIN_UP_DOWN.Visu_Adv_Arr[3] := FALSE;
   TL_PIN_UP_DOWN.Visu_Adv_Arr[4] := FALSE;
   TL_PIN_UP_DOWN.Visu_Adv_Arr[5] := FALSE;
   TL_PIN_UP_DOWN.Visu_Adv_Arr[6] := FALSE;
   TL_PIN_UP_DOWN.Visu_Adv_Arr[7] := FALSE;
   TL_PIN_UP_DOWN.Visu_Adv_Arr[8] := FALSE;
   TL_PIN_UP_DOWN.Visu_Adv_Arr[9] := FALSE;
   TL_PIN_UP_DOWN.Visu_Adv_Arr[10] := FALSE;
   TL_PIN_UP_DOWN.Visu_Adv_Arr[11] := FALSE;
   TL_PIN_UP_DOWN.Visu_Adv_Arr[12] := FALSE;
   TL_PIN_UP_DOWN.Visu_Adv_Arr[13] := FALSE;
   TL_PIN_UP_DOWN.Visu_Adv_Arr[14] := FALSE;
   TL_PIN_UP_DOWN.Visu_Adv_Arr[15] := FALSE;
   TL_PIN_UP_DOWN.Visu_Ret_Arr[0] := FALSE;
   TL_PIN_UP_DOWN.Visu_Ret_Arr[1] := FALSE;
   TL_PIN_UP_DOWN.Visu_Ret_Arr[2] := FALSE;
   TL_PIN_UP_DOWN.Visu_Ret_Arr[3] := FALSE;
   TL_PIN_UP_DOWN.Visu_Ret_Arr[4] := FALSE;
   TL_PIN_UP_DOWN.Visu_Ret_Arr[5] := FALSE;
   TL_PIN_UP_DOWN.Visu_Ret_Arr[6] := FALSE;
   TL_PIN_UP_DOWN.Visu_Ret_Arr[7] := FALSE;
   TL_PIN_UP_DOWN.Visu_Ret_Arr[8] := FALSE;
   TL_PIN_UP_DOWN.Visu_Ret_Arr[9] := FALSE;
   TL_PIN_UP_DOWN.Visu_Ret_Arr[10] := FALSE;
   TL_PIN_UP_DOWN.Visu_Ret_Arr[11] := FALSE;
   TL_PIN_UP_DOWN.Visu_Ret_Arr[12] := FALSE;
   TL_PIN_UP_DOWN.Visu_Ret_Arr[13] := FALSE;
   TL_PIN_UP_DOWN.Visu_Ret_Arr[14] := FALSE;
   TL_PIN_UP_DOWN.Visu_Ret_Arr[15] := FALSE;
   TL_PIN_UP_DOWN.BLK_Move_Ret := 0;
   TL_PIN_UP_DOWN.Enable := FALSE;
   TL_PIN_UP_DOWN.Adv_End := FALSE;
   TL_PIN_UP_DOWN.Ret_End := FALSE;
   TL_CLAMP1_SOL.Enable_Aux := FALSE;
   TL_CLAMP1_SOL.Adv_Amount := 0;
   TL_CLAMP1_SOL.Ret_Amount := 0;
   TL_CLAMP1_SOL.LS_Adv1 := FALSE;
   TL_CLAMP1_SOL.LS_Ret1 := FALSE;
   TL_CLAMP1_SOL.LS_Adv2 := FALSE;
   TL_CLAMP1_SOL.LS_Ret2 := FALSE;
   TL_CLAMP1_SOL.LS_Adv3 := FALSE;
   TL_CLAMP1_SOL.LS_Ret3 := FALSE;
   TL_CLAMP1_SOL.LS_Adv4 := FALSE;
   TL_CLAMP1_SOL.LS_Ret4 := FALSE;
   TL_CLAMP1_SOL.SOL_Adv := FALSE;
   TL_CLAMP1_SOL.SOL_Ret := FALSE;
   TL_CLAMP1_SOL.M_Ready := FALSE;
   TL_CLAMP1_SOL.T_CHK1 := T#0MS;
   TL_CLAMP1_SOL.T_CHK2 := T#0MS;
   TL_CLAMP1_SOL.PB_Lamp_CHK := FALSE;
   TL_CLAMP1_SOL.PB_Error_Rst := FALSE;
   TL_CLAMP1_SOL.M_FLICK := FALSE;
   TL_CLAMP1_SOL.M_Adv_Err := FALSE;
   TL_CLAMP1_SOL.M_Ret_Err := FALSE;
   TL_CLAMP1_SOL.LP_Adv := FALSE;
   TL_CLAMP1_SOL.LP_Ret := FALSE;
   TL_CLAMP1_SOL.Visu_Adv := W#16#0;
   TL_CLAMP1_SOL.Visu_Ret := W#16#0;
   TL_CLAMP1_SOL.Error_T1.IN := FALSE;
   TL_CLAMP1_SOL.Error_T1.PT := T#0MS;
   TL_CLAMP1_SOL.Error_T1.Q := FALSE;
   TL_CLAMP1_SOL.Error_T1.ET := T#0MS;
   TL_CLAMP1_SOL.Error_T1.STATE := B#16#0;
   TL_CLAMP1_SOL.Error_T1.STIME := T#0MS;
   TL_CLAMP1_SOL.Error_T1.ATIME := T#0MS;
   TL_CLAMP1_SOL.Error_T2.IN := FALSE;
   TL_CLAMP1_SOL.Error_T2.PT := T#0MS;
   TL_CLAMP1_SOL.Error_T2.Q := FALSE;
   TL_CLAMP1_SOL.Error_T2.ET := T#0MS;
   TL_CLAMP1_SOL.Error_T2.STATE := B#16#0;
   TL_CLAMP1_SOL.Error_T2.STIME := T#0MS;
   TL_CLAMP1_SOL.Error_T2.ATIME := T#0MS;
   TL_CLAMP1_SOL.CHK_Aux1 := FALSE;
   TL_CLAMP1_SOL.CHK_Aux2 := FALSE;
   TL_CLAMP1_SOL.Error_T1_DN := FALSE;
   TL_CLAMP1_SOL.Error_T2_DN := FALSE;
   TL_CLAMP1_SOL.Adv_Memo := FALSE;
   TL_CLAMP1_SOL.Visu_Adv_Arr[0] := FALSE;
   TL_CLAMP1_SOL.Visu_Adv_Arr[1] := FALSE;
   TL_CLAMP1_SOL.Visu_Adv_Arr[2] := FALSE;
   TL_CLAMP1_SOL.Visu_Adv_Arr[3] := FALSE;
   TL_CLAMP1_SOL.Visu_Adv_Arr[4] := FALSE;
   TL_CLAMP1_SOL.Visu_Adv_Arr[5] := FALSE;
   TL_CLAMP1_SOL.Visu_Adv_Arr[6] := FALSE;
   TL_CLAMP1_SOL.Visu_Adv_Arr[7] := FALSE;
   TL_CLAMP1_SOL.Visu_Adv_Arr[8] := FALSE;
   TL_CLAMP1_SOL.Visu_Adv_Arr[9] := FALSE;
   TL_CLAMP1_SOL.Visu_Adv_Arr[10] := FALSE;
   TL_CLAMP1_SOL.Visu_Adv_Arr[11] := FALSE;
   TL_CLAMP1_SOL.Visu_Adv_Arr[12] := FALSE;
   TL_CLAMP1_SOL.Visu_Adv_Arr[13] := FALSE;
   TL_CLAMP1_SOL.Visu_Adv_Arr[14] := FALSE;
   TL_CLAMP1_SOL.Visu_Adv_Arr[15] := FALSE;
   TL_CLAMP1_SOL.Visu_Ret_Arr[0] := FALSE;
   TL_CLAMP1_SOL.Visu_Ret_Arr[1] := FALSE;
   TL_CLAMP1_SOL.Visu_Ret_Arr[2] := FALSE;
   TL_CLAMP1_SOL.Visu_Ret_Arr[3] := FALSE;
   TL_CLAMP1_SOL.Visu_Ret_Arr[4] := FALSE;
   TL_CLAMP1_SOL.Visu_Ret_Arr[5] := FALSE;
   TL_CLAMP1_SOL.Visu_Ret_Arr[6] := FALSE;
   TL_CLAMP1_SOL.Visu_Ret_Arr[7] := FALSE;
   TL_CLAMP1_SOL.Visu_Ret_Arr[8] := FALSE;
   TL_CLAMP1_SOL.Visu_Ret_Arr[9] := FALSE;
   TL_CLAMP1_SOL.Visu_Ret_Arr[10] := FALSE;
   TL_CLAMP1_SOL.Visu_Ret_Arr[11] := FALSE;
   TL_CLAMP1_SOL.Visu_Ret_Arr[12] := FALSE;
   TL_CLAMP1_SOL.Visu_Ret_Arr[13] := FALSE;
   TL_CLAMP1_SOL.Visu_Ret_Arr[14] := FALSE;
   TL_CLAMP1_SOL.Visu_Ret_Arr[15] := FALSE;
   TL_CLAMP1_SOL.BLK_Move_Ret := 0;
   TL_CLAMP1_SOL.Enable := FALSE;
   TL_CLAMP1_SOL.Adv_End := FALSE;
   TL_CLAMP1_SOL.Ret_End := FALSE;
   TL_CLAMP2_SOL.Enable_Aux := FALSE;
   TL_CLAMP2_SOL.Adv_Amount := 0;
   TL_CLAMP2_SOL.Ret_Amount := 0;
   TL_CLAMP2_SOL.LS_Adv1 := FALSE;
   TL_CLAMP2_SOL.LS_Ret1 := FALSE;
   TL_CLAMP2_SOL.LS_Adv2 := FALSE;
   TL_CLAMP2_SOL.LS_Ret2 := FALSE;
   TL_CLAMP2_SOL.LS_Adv3 := FALSE;
   TL_CLAMP2_SOL.LS_Ret3 := FALSE;
   TL_CLAMP2_SOL.LS_Adv4 := FALSE;
   TL_CLAMP2_SOL.LS_Ret4 := FALSE;
   TL_CLAMP2_SOL.SOL_Adv := FALSE;
   TL_CLAMP2_SOL.SOL_Ret := FALSE;
   TL_CLAMP2_SOL.M_Ready := FALSE;
   TL_CLAMP2_SOL.T_CHK1 := T#0MS;
   TL_CLAMP2_SOL.T_CHK2 := T#0MS;
   TL_CLAMP2_SOL.PB_Lamp_CHK := FALSE;
   TL_CLAMP2_SOL.PB_Error_Rst := FALSE;
   TL_CLAMP2_SOL.M_FLICK := FALSE;
   TL_CLAMP2_SOL.M_Adv_Err := FALSE;
   TL_CLAMP2_SOL.M_Ret_Err := FALSE;
   TL_CLAMP2_SOL.LP_Adv := FALSE;
   TL_CLAMP2_SOL.LP_Ret := FALSE;
   TL_CLAMP2_SOL.Visu_Adv := W#16#0;
   TL_CLAMP2_SOL.Visu_Ret := W#16#0;
   TL_CLAMP2_SOL.Error_T1.IN := FALSE;
   TL_CLAMP2_SOL.Error_T1.PT := T#0MS;
   TL_CLAMP2_SOL.Error_T1.Q := FALSE;
   TL_CLAMP2_SOL.Error_T1.ET := T#0MS;
   TL_CLAMP2_SOL.Error_T1.STATE := B#16#0;
   TL_CLAMP2_SOL.Error_T1.STIME := T#0MS;
   TL_CLAMP2_SOL.Error_T1.ATIME := T#0MS;
   TL_CLAMP2_SOL.Error_T2.IN := FALSE;
   TL_CLAMP2_SOL.Error_T2.PT := T#0MS;
   TL_CLAMP2_SOL.Error_T2.Q := FALSE;
   TL_CLAMP2_SOL.Error_T2.ET := T#0MS;
   TL_CLAMP2_SOL.Error_T2.STATE := B#16#0;
   TL_CLAMP2_SOL.Error_T2.STIME := T#0MS;
   TL_CLAMP2_SOL.Error_T2.ATIME := T#0MS;
   TL_CLAMP2_SOL.CHK_Aux1 := FALSE;
   TL_CLAMP2_SOL.CHK_Aux2 := FALSE;
   TL_CLAMP2_SOL.Error_T1_DN := FALSE;
   TL_CLAMP2_SOL.Error_T2_DN := FALSE;
   TL_CLAMP2_SOL.Adv_Memo := FALSE;
   TL_CLAMP2_SOL.Visu_Adv_Arr[0] := FALSE;
   TL_CLAMP2_SOL.Visu_Adv_Arr[1] := FALSE;
   TL_CLAMP2_SOL.Visu_Adv_Arr[2] := FALSE;
   TL_CLAMP2_SOL.Visu_Adv_Arr[3] := FALSE;
   TL_CLAMP2_SOL.Visu_Adv_Arr[4] := FALSE;
   TL_CLAMP2_SOL.Visu_Adv_Arr[5] := FALSE;
   TL_CLAMP2_SOL.Visu_Adv_Arr[6] := FALSE;
   TL_CLAMP2_SOL.Visu_Adv_Arr[7] := FALSE;
   TL_CLAMP2_SOL.Visu_Adv_Arr[8] := FALSE;
   TL_CLAMP2_SOL.Visu_Adv_Arr[9] := FALSE;
   TL_CLAMP2_SOL.Visu_Adv_Arr[10] := FALSE;
   TL_CLAMP2_SOL.Visu_Adv_Arr[11] := FALSE;
   TL_CLAMP2_SOL.Visu_Adv_Arr[12] := FALSE;
   TL_CLAMP2_SOL.Visu_Adv_Arr[13] := FALSE;
   TL_CLAMP2_SOL.Visu_Adv_Arr[14] := FALSE;
   TL_CLAMP2_SOL.Visu_Adv_Arr[15] := FALSE;
   TL_CLAMP2_SOL.Visu_Ret_Arr[0] := FALSE;
   TL_CLAMP2_SOL.Visu_Ret_Arr[1] := FALSE;
   TL_CLAMP2_SOL.Visu_Ret_Arr[2] := FALSE;
   TL_CLAMP2_SOL.Visu_Ret_Arr[3] := FALSE;
   TL_CLAMP2_SOL.Visu_Ret_Arr[4] := FALSE;
   TL_CLAMP2_SOL.Visu_Ret_Arr[5] := FALSE;
   TL_CLAMP2_SOL.Visu_Ret_Arr[6] := FALSE;
   TL_CLAMP2_SOL.Visu_Ret_Arr[7] := FALSE;
   TL_CLAMP2_SOL.Visu_Ret_Arr[8] := FALSE;
   TL_CLAMP2_SOL.Visu_Ret_Arr[9] := FALSE;
   TL_CLAMP2_SOL.Visu_Ret_Arr[10] := FALSE;
   TL_CLAMP2_SOL.Visu_Ret_Arr[11] := FALSE;
   TL_CLAMP2_SOL.Visu_Ret_Arr[12] := FALSE;
   TL_CLAMP2_SOL.Visu_Ret_Arr[13] := FALSE;
   TL_CLAMP2_SOL.Visu_Ret_Arr[14] := FALSE;
   TL_CLAMP2_SOL.Visu_Ret_Arr[15] := FALSE;
   TL_CLAMP2_SOL.BLK_Move_Ret := 0;
   TL_CLAMP2_SOL.Enable := FALSE;
   TL_CLAMP2_SOL.Adv_End := FALSE;
   TL_CLAMP2_SOL.Ret_End := FALSE;
   TL_GUN1_SHIFT.Enable_Aux := FALSE;
   TL_GUN1_SHIFT.Adv_Amount := 0;
   TL_GUN1_SHIFT.Ret_Amount := 0;
   TL_GUN1_SHIFT.LS_Adv1 := FALSE;
   TL_GUN1_SHIFT.LS_Ret1 := FALSE;
   TL_GUN1_SHIFT.LS_Adv2 := FALSE;
   TL_GUN1_SHIFT.LS_Ret2 := FALSE;
   TL_GUN1_SHIFT.LS_Adv3 := FALSE;
   TL_GUN1_SHIFT.LS_Ret3 := FALSE;
   TL_GUN1_SHIFT.LS_Adv4 := FALSE;
   TL_GUN1_SHIFT.LS_Ret4 := FALSE;
   TL_GUN1_SHIFT.SOL_Adv := FALSE;
   TL_GUN1_SHIFT.SOL_Ret := FALSE;
   TL_GUN1_SHIFT.M_Ready := FALSE;
   TL_GUN1_SHIFT.T_CHK1 := T#0MS;
   TL_GUN1_SHIFT.T_CHK2 := T#0MS;
   TL_GUN1_SHIFT.PB_Lamp_CHK := FALSE;
   TL_GUN1_SHIFT.PB_Error_Rst := FALSE;
   TL_GUN1_SHIFT.M_FLICK := FALSE;
   TL_GUN1_SHIFT.M_Adv_Err := FALSE;
   TL_GUN1_SHIFT.M_Ret_Err := FALSE;
   TL_GUN1_SHIFT.LP_Adv := FALSE;
   TL_GUN1_SHIFT.LP_Ret := FALSE;
   TL_GUN1_SHIFT.Visu_Adv := W#16#0;
   TL_GUN1_SHIFT.Visu_Ret := W#16#0;
   TL_GUN1_SHIFT.Error_T1.IN := FALSE;
   TL_GUN1_SHIFT.Error_T1.PT := T#0MS;
   TL_GUN1_SHIFT.Error_T1.Q := FALSE;
   TL_GUN1_SHIFT.Error_T1.ET := T#0MS;
   TL_GUN1_SHIFT.Error_T1.STATE := B#16#0;
   TL_GUN1_SHIFT.Error_T1.STIME := T#0MS;
   TL_GUN1_SHIFT.Error_T1.ATIME := T#0MS;
   TL_GUN1_SHIFT.Error_T2.IN := FALSE;
   TL_GUN1_SHIFT.Error_T2.PT := T#0MS;
   TL_GUN1_SHIFT.Error_T2.Q := FALSE;
   TL_GUN1_SHIFT.Error_T2.ET := T#0MS;
   TL_GUN1_SHIFT.Error_T2.STATE := B#16#0;
   TL_GUN1_SHIFT.Error_T2.STIME := T#0MS;
   TL_GUN1_SHIFT.Error_T2.ATIME := T#0MS;
   TL_GUN1_SHIFT.CHK_Aux1 := FALSE;
   TL_GUN1_SHIFT.CHK_Aux2 := FALSE;
   TL_GUN1_SHIFT.Error_T1_DN := FALSE;
   TL_GUN1_SHIFT.Error_T2_DN := FALSE;
   TL_GUN1_SHIFT.Adv_Memo := FALSE;
   TL_GUN1_SHIFT.Visu_Adv_Arr[0] := FALSE;
   TL_GUN1_SHIFT.Visu_Adv_Arr[1] := FALSE;
   TL_GUN1_SHIFT.Visu_Adv_Arr[2] := FALSE;
   TL_GUN1_SHIFT.Visu_Adv_Arr[3] := FALSE;
   TL_GUN1_SHIFT.Visu_Adv_Arr[4] := FALSE;
   TL_GUN1_SHIFT.Visu_Adv_Arr[5] := FALSE;
   TL_GUN1_SHIFT.Visu_Adv_Arr[6] := FALSE;
   TL_GUN1_SHIFT.Visu_Adv_Arr[7] := FALSE;
   TL_GUN1_SHIFT.Visu_Adv_Arr[8] := FALSE;
   TL_GUN1_SHIFT.Visu_Adv_Arr[9] := FALSE;
   TL_GUN1_SHIFT.Visu_Adv_Arr[10] := FALSE;
   TL_GUN1_SHIFT.Visu_Adv_Arr[11] := FALSE;
   TL_GUN1_SHIFT.Visu_Adv_Arr[12] := FALSE;
   TL_GUN1_SHIFT.Visu_Adv_Arr[13] := FALSE;
   TL_GUN1_SHIFT.Visu_Adv_Arr[14] := FALSE;
   TL_GUN1_SHIFT.Visu_Adv_Arr[15] := FALSE;
   TL_GUN1_SHIFT.Visu_Ret_Arr[0] := FALSE;
   TL_GUN1_SHIFT.Visu_Ret_Arr[1] := FALSE;
   TL_GUN1_SHIFT.Visu_Ret_Arr[2] := FALSE;
   TL_GUN1_SHIFT.Visu_Ret_Arr[3] := FALSE;
   TL_GUN1_SHIFT.Visu_Ret_Arr[4] := FALSE;
   TL_GUN1_SHIFT.Visu_Ret_Arr[5] := FALSE;
   TL_GUN1_SHIFT.Visu_Ret_Arr[6] := FALSE;
   TL_GUN1_SHIFT.Visu_Ret_Arr[7] := FALSE;
   TL_GUN1_SHIFT.Visu_Ret_Arr[8] := FALSE;
   TL_GUN1_SHIFT.Visu_Ret_Arr[9] := FALSE;
   TL_GUN1_SHIFT.Visu_Ret_Arr[10] := FALSE;
   TL_GUN1_SHIFT.Visu_Ret_Arr[11] := FALSE;
   TL_GUN1_SHIFT.Visu_Ret_Arr[12] := FALSE;
   TL_GUN1_SHIFT.Visu_Ret_Arr[13] := FALSE;
   TL_GUN1_SHIFT.Visu_Ret_Arr[14] := FALSE;
   TL_GUN1_SHIFT.Visu_Ret_Arr[15] := FALSE;
   TL_GUN1_SHIFT.BLK_Move_Ret := 0;
   TL_GUN1_SHIFT.Enable := FALSE;
   TL_GUN1_SHIFT.Adv_End := FALSE;
   TL_GUN1_SHIFT.Ret_End := FALSE;
   TL_GUN2_SHIFT.Enable_Aux := FALSE;
   TL_GUN2_SHIFT.Adv_Amount := 0;
   TL_GUN2_SHIFT.Ret_Amount := 0;
   TL_GUN2_SHIFT.LS_Adv1 := FALSE;
   TL_GUN2_SHIFT.LS_Ret1 := FALSE;
   TL_GUN2_SHIFT.LS_Adv2 := FALSE;
   TL_GUN2_SHIFT.LS_Ret2 := FALSE;
   TL_GUN2_SHIFT.LS_Adv3 := FALSE;
   TL_GUN2_SHIFT.LS_Ret3 := FALSE;
   TL_GUN2_SHIFT.LS_Adv4 := FALSE;
   TL_GUN2_SHIFT.LS_Ret4 := FALSE;
   TL_GUN2_SHIFT.SOL_Adv := FALSE;
   TL_GUN2_SHIFT.SOL_Ret := FALSE;
   TL_GUN2_SHIFT.M_Ready := FALSE;
   TL_GUN2_SHIFT.T_CHK1 := T#0MS;
   TL_GUN2_SHIFT.T_CHK2 := T#0MS;
   TL_GUN2_SHIFT.PB_Lamp_CHK := FALSE;
   TL_GUN2_SHIFT.PB_Error_Rst := FALSE;
   TL_GUN2_SHIFT.M_FLICK := FALSE;
   TL_GUN2_SHIFT.M_Adv_Err := FALSE;
   TL_GUN2_SHIFT.M_Ret_Err := FALSE;
   TL_GUN2_SHIFT.LP_Adv := FALSE;
   TL_GUN2_SHIFT.LP_Ret := FALSE;
   TL_GUN2_SHIFT.Visu_Adv := W#16#0;
   TL_GUN2_SHIFT.Visu_Ret := W#16#0;
   TL_GUN2_SHIFT.Error_T1.IN := FALSE;
   TL_GUN2_SHIFT.Error_T1.PT := T#0MS;
   TL_GUN2_SHIFT.Error_T1.Q := FALSE;
   TL_GUN2_SHIFT.Error_T1.ET := T#0MS;
   TL_GUN2_SHIFT.Error_T1.STATE := B#16#0;
   TL_GUN2_SHIFT.Error_T1.STIME := T#0MS;
   TL_GUN2_SHIFT.Error_T1.ATIME := T#0MS;
   TL_GUN2_SHIFT.Error_T2.IN := FALSE;
   TL_GUN2_SHIFT.Error_T2.PT := T#0MS;
   TL_GUN2_SHIFT.Error_T2.Q := FALSE;
   TL_GUN2_SHIFT.Error_T2.ET := T#0MS;
   TL_GUN2_SHIFT.Error_T2.STATE := B#16#0;
   TL_GUN2_SHIFT.Error_T2.STIME := T#0MS;
   TL_GUN2_SHIFT.Error_T2.ATIME := T#0MS;
   TL_GUN2_SHIFT.CHK_Aux1 := FALSE;
   TL_GUN2_SHIFT.CHK_Aux2 := FALSE;
   TL_GUN2_SHIFT.Error_T1_DN := FALSE;
   TL_GUN2_SHIFT.Error_T2_DN := FALSE;
   TL_GUN2_SHIFT.Adv_Memo := FALSE;
   TL_GUN2_SHIFT.Visu_Adv_Arr[0] := FALSE;
   TL_GUN2_SHIFT.Visu_Adv_Arr[1] := FALSE;
   TL_GUN2_SHIFT.Visu_Adv_Arr[2] := FALSE;
   TL_GUN2_SHIFT.Visu_Adv_Arr[3] := FALSE;
   TL_GUN2_SHIFT.Visu_Adv_Arr[4] := FALSE;
   TL_GUN2_SHIFT.Visu_Adv_Arr[5] := FALSE;
   TL_GUN2_SHIFT.Visu_Adv_Arr[6] := FALSE;
   TL_GUN2_SHIFT.Visu_Adv_Arr[7] := FALSE;
   TL_GUN2_SHIFT.Visu_Adv_Arr[8] := FALSE;
   TL_GUN2_SHIFT.Visu_Adv_Arr[9] := FALSE;
   TL_GUN2_SHIFT.Visu_Adv_Arr[10] := FALSE;
   TL_GUN2_SHIFT.Visu_Adv_Arr[11] := FALSE;
   TL_GUN2_SHIFT.Visu_Adv_Arr[12] := FALSE;
   TL_GUN2_SHIFT.Visu_Adv_Arr[13] := FALSE;
   TL_GUN2_SHIFT.Visu_Adv_Arr[14] := FALSE;
   TL_GUN2_SHIFT.Visu_Adv_Arr[15] := FALSE;
   TL_GUN2_SHIFT.Visu_Ret_Arr[0] := FALSE;
   TL_GUN2_SHIFT.Visu_Ret_Arr[1] := FALSE;
   TL_GUN2_SHIFT.Visu_Ret_Arr[2] := FALSE;
   TL_GUN2_SHIFT.Visu_Ret_Arr[3] := FALSE;
   TL_GUN2_SHIFT.Visu_Ret_Arr[4] := FALSE;
   TL_GUN2_SHIFT.Visu_Ret_Arr[5] := FALSE;
   TL_GUN2_SHIFT.Visu_Ret_Arr[6] := FALSE;
   TL_GUN2_SHIFT.Visu_Ret_Arr[7] := FALSE;
   TL_GUN2_SHIFT.Visu_Ret_Arr[8] := FALSE;
   TL_GUN2_SHIFT.Visu_Ret_Arr[9] := FALSE;
   TL_GUN2_SHIFT.Visu_Ret_Arr[10] := FALSE;
   TL_GUN2_SHIFT.Visu_Ret_Arr[11] := FALSE;
   TL_GUN2_SHIFT.Visu_Ret_Arr[12] := FALSE;
   TL_GUN2_SHIFT.Visu_Ret_Arr[13] := FALSE;
   TL_GUN2_SHIFT.Visu_Ret_Arr[14] := FALSE;
   TL_GUN2_SHIFT.Visu_Ret_Arr[15] := FALSE;
   TL_GUN2_SHIFT.BLK_Move_Ret := 0;
   TL_GUN2_SHIFT.Enable := FALSE;
   TL_GUN2_SHIFT.Adv_End := FALSE;
   TL_GUN2_SHIFT.Ret_End := FALSE;
   TL_GUN3_1_SHIFT.Enable_Aux := FALSE;
   TL_GUN3_1_SHIFT.Adv_Amount := 0;
   TL_GUN3_1_SHIFT.Ret_Amount := 0;
   TL_GUN3_1_SHIFT.LS_Adv1 := FALSE;
   TL_GUN3_1_SHIFT.LS_Ret1 := FALSE;
   TL_GUN3_1_SHIFT.LS_Adv2 := FALSE;
   TL_GUN3_1_SHIFT.LS_Ret2 := FALSE;
   TL_GUN3_1_SHIFT.LS_Adv3 := FALSE;
   TL_GUN3_1_SHIFT.LS_Ret3 := FALSE;
   TL_GUN3_1_SHIFT.LS_Adv4 := FALSE;
   TL_GUN3_1_SHIFT.LS_Ret4 := FALSE;
   TL_GUN3_1_SHIFT.SOL_Adv := FALSE;
   TL_GUN3_1_SHIFT.SOL_Ret := FALSE;
   TL_GUN3_1_SHIFT.M_Ready := FALSE;
   TL_GUN3_1_SHIFT.T_CHK1 := T#0MS;
   TL_GUN3_1_SHIFT.T_CHK2 := T#0MS;
   TL_GUN3_1_SHIFT.PB_Lamp_CHK := FALSE;
   TL_GUN3_1_SHIFT.PB_Error_Rst := FALSE;
   TL_GUN3_1_SHIFT.M_FLICK := FALSE;
   TL_GUN3_1_SHIFT.M_Adv_Err := FALSE;
   TL_GUN3_1_SHIFT.M_Ret_Err := FALSE;
   TL_GUN3_1_SHIFT.LP_Adv := FALSE;
   TL_GUN3_1_SHIFT.LP_Ret := FALSE;
   TL_GUN3_1_SHIFT.Visu_Adv := W#16#0;
   TL_GUN3_1_SHIFT.Visu_Ret := W#16#0;
   TL_GUN3_1_SHIFT.Error_T1.IN := FALSE;
   TL_GUN3_1_SHIFT.Error_T1.PT := T#0MS;
   TL_GUN3_1_SHIFT.Error_T1.Q := FALSE;
   TL_GUN3_1_SHIFT.Error_T1.ET := T#0MS;
   TL_GUN3_1_SHIFT.Error_T1.STATE := B#16#0;
   TL_GUN3_1_SHIFT.Error_T1.STIME := T#0MS;
   TL_GUN3_1_SHIFT.Error_T1.ATIME := T#0MS;
   TL_GUN3_1_SHIFT.Error_T2.IN := FALSE;
   TL_GUN3_1_SHIFT.Error_T2.PT := T#0MS;
   TL_GUN3_1_SHIFT.Error_T2.Q := FALSE;
   TL_GUN3_1_SHIFT.Error_T2.ET := T#0MS;
   TL_GUN3_1_SHIFT.Error_T2.STATE := B#16#0;
   TL_GUN3_1_SHIFT.Error_T2.STIME := T#0MS;
   TL_GUN3_1_SHIFT.Error_T2.ATIME := T#0MS;
   TL_GUN3_1_SHIFT.CHK_Aux1 := FALSE;
   TL_GUN3_1_SHIFT.CHK_Aux2 := FALSE;
   TL_GUN3_1_SHIFT.Error_T1_DN := FALSE;
   TL_GUN3_1_SHIFT.Error_T2_DN := FALSE;
   TL_GUN3_1_SHIFT.Adv_Memo := FALSE;
   TL_GUN3_1_SHIFT.Visu_Adv_Arr[0] := FALSE;
   TL_GUN3_1_SHIFT.Visu_Adv_Arr[1] := FALSE;
   TL_GUN3_1_SHIFT.Visu_Adv_Arr[2] := FALSE;
   TL_GUN3_1_SHIFT.Visu_Adv_Arr[3] := FALSE;
   TL_GUN3_1_SHIFT.Visu_Adv_Arr[4] := FALSE;
   TL_GUN3_1_SHIFT.Visu_Adv_Arr[5] := FALSE;
   TL_GUN3_1_SHIFT.Visu_Adv_Arr[6] := FALSE;
   TL_GUN3_1_SHIFT.Visu_Adv_Arr[7] := FALSE;
   TL_GUN3_1_SHIFT.Visu_Adv_Arr[8] := FALSE;
   TL_GUN3_1_SHIFT.Visu_Adv_Arr[9] := FALSE;
   TL_GUN3_1_SHIFT.Visu_Adv_Arr[10] := FALSE;
   TL_GUN3_1_SHIFT.Visu_Adv_Arr[11] := FALSE;
   TL_GUN3_1_SHIFT.Visu_Adv_Arr[12] := FALSE;
   TL_GUN3_1_SHIFT.Visu_Adv_Arr[13] := FALSE;
   TL_GUN3_1_SHIFT.Visu_Adv_Arr[14] := FALSE;
   TL_GUN3_1_SHIFT.Visu_Adv_Arr[15] := FALSE;
   TL_GUN3_1_SHIFT.Visu_Ret_Arr[0] := FALSE;
   TL_GUN3_1_SHIFT.Visu_Ret_Arr[1] := FALSE;
   TL_GUN3_1_SHIFT.Visu_Ret_Arr[2] := FALSE;
   TL_GUN3_1_SHIFT.Visu_Ret_Arr[3] := FALSE;
   TL_GUN3_1_SHIFT.Visu_Ret_Arr[4] := FALSE;
   TL_GUN3_1_SHIFT.Visu_Ret_Arr[5] := FALSE;
   TL_GUN3_1_SHIFT.Visu_Ret_Arr[6] := FALSE;
   TL_GUN3_1_SHIFT.Visu_Ret_Arr[7] := FALSE;
   TL_GUN3_1_SHIFT.Visu_Ret_Arr[8] := FALSE;
   TL_GUN3_1_SHIFT.Visu_Ret_Arr[9] := FALSE;
   TL_GUN3_1_SHIFT.Visu_Ret_Arr[10] := FALSE;
   TL_GUN3_1_SHIFT.Visu_Ret_Arr[11] := FALSE;
   TL_GUN3_1_SHIFT.Visu_Ret_Arr[12] := FALSE;
   TL_GUN3_1_SHIFT.Visu_Ret_Arr[13] := FALSE;
   TL_GUN3_1_SHIFT.Visu_Ret_Arr[14] := FALSE;
   TL_GUN3_1_SHIFT.Visu_Ret_Arr[15] := FALSE;
   TL_GUN3_1_SHIFT.BLK_Move_Ret := 0;
   TL_GUN3_1_SHIFT.Enable := FALSE;
   TL_GUN3_1_SHIFT.Adv_End := FALSE;
   TL_GUN3_1_SHIFT.Ret_End := FALSE;
   TL_GUN3_2_SHIFT.Enable_Aux := FALSE;
   TL_GUN3_2_SHIFT.Adv_Amount := 0;
   TL_GUN3_2_SHIFT.Ret_Amount := 0;
   TL_GUN3_2_SHIFT.LS_Adv1 := FALSE;
   TL_GUN3_2_SHIFT.LS_Ret1 := FALSE;
   TL_GUN3_2_SHIFT.LS_Adv2 := FALSE;
   TL_GUN3_2_SHIFT.LS_Ret2 := FALSE;
   TL_GUN3_2_SHIFT.LS_Adv3 := FALSE;
   TL_GUN3_2_SHIFT.LS_Ret3 := FALSE;
   TL_GUN3_2_SHIFT.LS_Adv4 := FALSE;
   TL_GUN3_2_SHIFT.LS_Ret4 := FALSE;
   TL_GUN3_2_SHIFT.SOL_Adv := FALSE;
   TL_GUN3_2_SHIFT.SOL_Ret := FALSE;
   TL_GUN3_2_SHIFT.M_Ready := FALSE;
   TL_GUN3_2_SHIFT.T_CHK1 := T#0MS;
   TL_GUN3_2_SHIFT.T_CHK2 := T#0MS;
   TL_GUN3_2_SHIFT.PB_Lamp_CHK := FALSE;
   TL_GUN3_2_SHIFT.PB_Error_Rst := FALSE;
   TL_GUN3_2_SHIFT.M_FLICK := FALSE;
   TL_GUN3_2_SHIFT.M_Adv_Err := FALSE;
   TL_GUN3_2_SHIFT.M_Ret_Err := FALSE;
   TL_GUN3_2_SHIFT.LP_Adv := FALSE;
   TL_GUN3_2_SHIFT.LP_Ret := FALSE;
   TL_GUN3_2_SHIFT.Visu_Adv := W#16#0;
   TL_GUN3_2_SHIFT.Visu_Ret := W#16#0;
   TL_GUN3_2_SHIFT.Error_T1.IN := FALSE;
   TL_GUN3_2_SHIFT.Error_T1.PT := T#0MS;
   TL_GUN3_2_SHIFT.Error_T1.Q := FALSE;
   TL_GUN3_2_SHIFT.Error_T1.ET := T#0MS;
   TL_GUN3_2_SHIFT.Error_T1.STATE := B#16#0;
   TL_GUN3_2_SHIFT.Error_T1.STIME := T#0MS;
   TL_GUN3_2_SHIFT.Error_T1.ATIME := T#0MS;
   TL_GUN3_2_SHIFT.Error_T2.IN := FALSE;
   TL_GUN3_2_SHIFT.Error_T2.PT := T#0MS;
   TL_GUN3_2_SHIFT.Error_T2.Q := FALSE;
   TL_GUN3_2_SHIFT.Error_T2.ET := T#0MS;
   TL_GUN3_2_SHIFT.Error_T2.STATE := B#16#0;
   TL_GUN3_2_SHIFT.Error_T2.STIME := T#0MS;
   TL_GUN3_2_SHIFT.Error_T2.ATIME := T#0MS;
   TL_GUN3_2_SHIFT.CHK_Aux1 := FALSE;
   TL_GUN3_2_SHIFT.CHK_Aux2 := FALSE;
   TL_GUN3_2_SHIFT.Error_T1_DN := FALSE;
   TL_GUN3_2_SHIFT.Error_T2_DN := FALSE;
   TL_GUN3_2_SHIFT.Adv_Memo := FALSE;
   TL_GUN3_2_SHIFT.Visu_Adv_Arr[0] := FALSE;
   TL_GUN3_2_SHIFT.Visu_Adv_Arr[1] := FALSE;
   TL_GUN3_2_SHIFT.Visu_Adv_Arr[2] := FALSE;
   TL_GUN3_2_SHIFT.Visu_Adv_Arr[3] := FALSE;
   TL_GUN3_2_SHIFT.Visu_Adv_Arr[4] := FALSE;
   TL_GUN3_2_SHIFT.Visu_Adv_Arr[5] := FALSE;
   TL_GUN3_2_SHIFT.Visu_Adv_Arr[6] := FALSE;
   TL_GUN3_2_SHIFT.Visu_Adv_Arr[7] := FALSE;
   TL_GUN3_2_SHIFT.Visu_Adv_Arr[8] := FALSE;
   TL_GUN3_2_SHIFT.Visu_Adv_Arr[9] := FALSE;
   TL_GUN3_2_SHIFT.Visu_Adv_Arr[10] := FALSE;
   TL_GUN3_2_SHIFT.Visu_Adv_Arr[11] := FALSE;
   TL_GUN3_2_SHIFT.Visu_Adv_Arr[12] := FALSE;
   TL_GUN3_2_SHIFT.Visu_Adv_Arr[13] := FALSE;
   TL_GUN3_2_SHIFT.Visu_Adv_Arr[14] := FALSE;
   TL_GUN3_2_SHIFT.Visu_Adv_Arr[15] := FALSE;
   TL_GUN3_2_SHIFT.Visu_Ret_Arr[0] := FALSE;
   TL_GUN3_2_SHIFT.Visu_Ret_Arr[1] := FALSE;
   TL_GUN3_2_SHIFT.Visu_Ret_Arr[2] := FALSE;
   TL_GUN3_2_SHIFT.Visu_Ret_Arr[3] := FALSE;
   TL_GUN3_2_SHIFT.Visu_Ret_Arr[4] := FALSE;
   TL_GUN3_2_SHIFT.Visu_Ret_Arr[5] := FALSE;
   TL_GUN3_2_SHIFT.Visu_Ret_Arr[6] := FALSE;
   TL_GUN3_2_SHIFT.Visu_Ret_Arr[7] := FALSE;
   TL_GUN3_2_SHIFT.Visu_Ret_Arr[8] := FALSE;
   TL_GUN3_2_SHIFT.Visu_Ret_Arr[9] := FALSE;
   TL_GUN3_2_SHIFT.Visu_Ret_Arr[10] := FALSE;
   TL_GUN3_2_SHIFT.Visu_Ret_Arr[11] := FALSE;
   TL_GUN3_2_SHIFT.Visu_Ret_Arr[12] := FALSE;
   TL_GUN3_2_SHIFT.Visu_Ret_Arr[13] := FALSE;
   TL_GUN3_2_SHIFT.Visu_Ret_Arr[14] := FALSE;
   TL_GUN3_2_SHIFT.Visu_Ret_Arr[15] := FALSE;
   TL_GUN3_2_SHIFT.BLK_Move_Ret := 0;
   TL_GUN3_2_SHIFT.Enable := FALSE;
   TL_GUN3_2_SHIFT.Adv_End := FALSE;
   TL_GUN3_2_SHIFT.Ret_End := FALSE;
   LM_IDLE_LATCH.Enable_Aux := FALSE;
   LM_IDLE_LATCH.Adv_Amount := 0;
   LM_IDLE_LATCH.Ret_Amount := 0;
   LM_IDLE_LATCH.LS_Adv1 := FALSE;
   LM_IDLE_LATCH.LS_Ret1 := FALSE;
   LM_IDLE_LATCH.LS_Adv2 := FALSE;
   LM_IDLE_LATCH.LS_Ret2 := FALSE;
   LM_IDLE_LATCH.LS_Adv3 := FALSE;
   LM_IDLE_LATCH.LS_Ret3 := FALSE;
   LM_IDLE_LATCH.LS_Adv4 := FALSE;
   LM_IDLE_LATCH.LS_Ret4 := FALSE;
   LM_IDLE_LATCH.SOL_Adv := FALSE;
   LM_IDLE_LATCH.SOL_Ret := FALSE;
   LM_IDLE_LATCH.M_Ready := FALSE;
   LM_IDLE_LATCH.T_CHK1 := T#0MS;
   LM_IDLE_LATCH.T_CHK2 := T#0MS;
   LM_IDLE_LATCH.PB_Lamp_CHK := FALSE;
   LM_IDLE_LATCH.PB_Error_Rst := FALSE;
   LM_IDLE_LATCH.M_FLICK := FALSE;
   LM_IDLE_LATCH.M_Adv_Err := FALSE;
   LM_IDLE_LATCH.M_Ret_Err := FALSE;
   LM_IDLE_LATCH.LP_Adv := FALSE;
   LM_IDLE_LATCH.LP_Ret := FALSE;
   LM_IDLE_LATCH.Visu_Adv := W#16#0;
   LM_IDLE_LATCH.Visu_Ret := W#16#0;
   LM_IDLE_LATCH.Error_T1.IN := FALSE;
   LM_IDLE_LATCH.Error_T1.PT := T#0MS;
   LM_IDLE_LATCH.Error_T1.Q := FALSE;
   LM_IDLE_LATCH.Error_T1.ET := T#0MS;
   LM_IDLE_LATCH.Error_T1.STATE := B#16#0;
   LM_IDLE_LATCH.Error_T1.STIME := T#0MS;
   LM_IDLE_LATCH.Error_T1.ATIME := T#0MS;
   LM_IDLE_LATCH.Error_T2.IN := FALSE;
   LM_IDLE_LATCH.Error_T2.PT := T#0MS;
   LM_IDLE_LATCH.Error_T2.Q := FALSE;
   LM_IDLE_LATCH.Error_T2.ET := T#0MS;
   LM_IDLE_LATCH.Error_T2.STATE := B#16#0;
   LM_IDLE_LATCH.Error_T2.STIME := T#0MS;
   LM_IDLE_LATCH.Error_T2.ATIME := T#0MS;
   LM_IDLE_LATCH.CHK_Aux1 := FALSE;
   LM_IDLE_LATCH.CHK_Aux2 := FALSE;
   LM_IDLE_LATCH.Error_T1_DN := FALSE;
   LM_IDLE_LATCH.Error_T2_DN := FALSE;
   LM_IDLE_LATCH.Adv_Memo := FALSE;
   LM_IDLE_LATCH.Visu_Adv_Arr[0] := FALSE;
   LM_IDLE_LATCH.Visu_Adv_Arr[1] := FALSE;
   LM_IDLE_LATCH.Visu_Adv_Arr[2] := FALSE;
   LM_IDLE_LATCH.Visu_Adv_Arr[3] := FALSE;
   LM_IDLE_LATCH.Visu_Adv_Arr[4] := FALSE;
   LM_IDLE_LATCH.Visu_Adv_Arr[5] := FALSE;
   LM_IDLE_LATCH.Visu_Adv_Arr[6] := FALSE;
   LM_IDLE_LATCH.Visu_Adv_Arr[7] := FALSE;
   LM_IDLE_LATCH.Visu_Adv_Arr[8] := FALSE;
   LM_IDLE_LATCH.Visu_Adv_Arr[9] := FALSE;
   LM_IDLE_LATCH.Visu_Adv_Arr[10] := FALSE;
   LM_IDLE_LATCH.Visu_Adv_Arr[11] := FALSE;
   LM_IDLE_LATCH.Visu_Adv_Arr[12] := FALSE;
   LM_IDLE_LATCH.Visu_Adv_Arr[13] := FALSE;
   LM_IDLE_LATCH.Visu_Adv_Arr[14] := FALSE;
   LM_IDLE_LATCH.Visu_Adv_Arr[15] := FALSE;
   LM_IDLE_LATCH.Visu_Ret_Arr[0] := FALSE;
   LM_IDLE_LATCH.Visu_Ret_Arr[1] := FALSE;
   LM_IDLE_LATCH.Visu_Ret_Arr[2] := FALSE;
   LM_IDLE_LATCH.Visu_Ret_Arr[3] := FALSE;
   LM_IDLE_LATCH.Visu_Ret_Arr[4] := FALSE;
   LM_IDLE_LATCH.Visu_Ret_Arr[5] := FALSE;
   LM_IDLE_LATCH.Visu_Ret_Arr[6] := FALSE;
   LM_IDLE_LATCH.Visu_Ret_Arr[7] := FALSE;
   LM_IDLE_LATCH.Visu_Ret_Arr[8] := FALSE;
   LM_IDLE_LATCH.Visu_Ret_Arr[9] := FALSE;
   LM_IDLE_LATCH.Visu_Ret_Arr[10] := FALSE;
   LM_IDLE_LATCH.Visu_Ret_Arr[11] := FALSE;
   LM_IDLE_LATCH.Visu_Ret_Arr[12] := FALSE;
   LM_IDLE_LATCH.Visu_Ret_Arr[13] := FALSE;
   LM_IDLE_LATCH.Visu_Ret_Arr[14] := FALSE;
   LM_IDLE_LATCH.Visu_Ret_Arr[15] := FALSE;
   LM_IDLE_LATCH.BLK_Move_Ret := 0;
   LM_IDLE_LATCH.Enable := FALSE;
   LM_IDLE_LATCH.Adv_End := FALSE;
   LM_IDLE_LATCH.Ret_End := FALSE;
   TL_IDLE_LATCH.Enable_Aux := FALSE;
   TL_IDLE_LATCH.Adv_Amount := 0;
   TL_IDLE_LATCH.Ret_Amount := 0;
   TL_IDLE_LATCH.LS_Adv1 := FALSE;
   TL_IDLE_LATCH.LS_Ret1 := FALSE;
   TL_IDLE_LATCH.LS_Adv2 := FALSE;
   TL_IDLE_LATCH.LS_Ret2 := FALSE;
   TL_IDLE_LATCH.LS_Adv3 := FALSE;
   TL_IDLE_LATCH.LS_Ret3 := FALSE;
   TL_IDLE_LATCH.LS_Adv4 := FALSE;
   TL_IDLE_LATCH.LS_Ret4 := FALSE;
   TL_IDLE_LATCH.SOL_Adv := FALSE;
   TL_IDLE_LATCH.SOL_Ret := FALSE;
   TL_IDLE_LATCH.M_Ready := FALSE;
   TL_IDLE_LATCH.T_CHK1 := T#0MS;
   TL_IDLE_LATCH.T_CHK2 := T#0MS;
   TL_IDLE_LATCH.PB_Lamp_CHK := FALSE;
   TL_IDLE_LATCH.PB_Error_Rst := FALSE;
   TL_IDLE_LATCH.M_FLICK := FALSE;
   TL_IDLE_LATCH.M_Adv_Err := FALSE;
   TL_IDLE_LATCH.M_Ret_Err := FALSE;
   TL_IDLE_LATCH.LP_Adv := FALSE;
   TL_IDLE_LATCH.LP_Ret := FALSE;
   TL_IDLE_LATCH.Visu_Adv := W#16#0;
   TL_IDLE_LATCH.Visu_Ret := W#16#0;
   TL_IDLE_LATCH.Error_T1.IN := FALSE;
   TL_IDLE_LATCH.Error_T1.PT := T#0MS;
   TL_IDLE_LATCH.Error_T1.Q := FALSE;
   TL_IDLE_LATCH.Error_T1.ET := T#0MS;
   TL_IDLE_LATCH.Error_T1.STATE := B#16#0;
   TL_IDLE_LATCH.Error_T1.STIME := T#0MS;
   TL_IDLE_LATCH.Error_T1.ATIME := T#0MS;
   TL_IDLE_LATCH.Error_T2.IN := FALSE;
   TL_IDLE_LATCH.Error_T2.PT := T#0MS;
   TL_IDLE_LATCH.Error_T2.Q := FALSE;
   TL_IDLE_LATCH.Error_T2.ET := T#0MS;
   TL_IDLE_LATCH.Error_T2.STATE := B#16#0;
   TL_IDLE_LATCH.Error_T2.STIME := T#0MS;
   TL_IDLE_LATCH.Error_T2.ATIME := T#0MS;
   TL_IDLE_LATCH.CHK_Aux1 := FALSE;
   TL_IDLE_LATCH.CHK_Aux2 := FALSE;
   TL_IDLE_LATCH.Error_T1_DN := FALSE;
   TL_IDLE_LATCH.Error_T2_DN := FALSE;
   TL_IDLE_LATCH.Adv_Memo := FALSE;
   TL_IDLE_LATCH.Visu_Adv_Arr[0] := FALSE;
   TL_IDLE_LATCH.Visu_Adv_Arr[1] := FALSE;
   TL_IDLE_LATCH.Visu_Adv_Arr[2] := FALSE;
   TL_IDLE_LATCH.Visu_Adv_Arr[3] := FALSE;
   TL_IDLE_LATCH.Visu_Adv_Arr[4] := FALSE;
   TL_IDLE_LATCH.Visu_Adv_Arr[5] := FALSE;
   TL_IDLE_LATCH.Visu_Adv_Arr[6] := FALSE;
   TL_IDLE_LATCH.Visu_Adv_Arr[7] := FALSE;
   TL_IDLE_LATCH.Visu_Adv_Arr[8] := FALSE;
   TL_IDLE_LATCH.Visu_Adv_Arr[9] := FALSE;
   TL_IDLE_LATCH.Visu_Adv_Arr[10] := FALSE;
   TL_IDLE_LATCH.Visu_Adv_Arr[11] := FALSE;
   TL_IDLE_LATCH.Visu_Adv_Arr[12] := FALSE;
   TL_IDLE_LATCH.Visu_Adv_Arr[13] := FALSE;
   TL_IDLE_LATCH.Visu_Adv_Arr[14] := FALSE;
   TL_IDLE_LATCH.Visu_Adv_Arr[15] := FALSE;
   TL_IDLE_LATCH.Visu_Ret_Arr[0] := FALSE;
   TL_IDLE_LATCH.Visu_Ret_Arr[1] := FALSE;
   TL_IDLE_LATCH.Visu_Ret_Arr[2] := FALSE;
   TL_IDLE_LATCH.Visu_Ret_Arr[3] := FALSE;
   TL_IDLE_LATCH.Visu_Ret_Arr[4] := FALSE;
   TL_IDLE_LATCH.Visu_Ret_Arr[5] := FALSE;
   TL_IDLE_LATCH.Visu_Ret_Arr[6] := FALSE;
   TL_IDLE_LATCH.Visu_Ret_Arr[7] := FALSE;
   TL_IDLE_LATCH.Visu_Ret_Arr[8] := FALSE;
   TL_IDLE_LATCH.Visu_Ret_Arr[9] := FALSE;
   TL_IDLE_LATCH.Visu_Ret_Arr[10] := FALSE;
   TL_IDLE_LATCH.Visu_Ret_Arr[11] := FALSE;
   TL_IDLE_LATCH.Visu_Ret_Arr[12] := FALSE;
   TL_IDLE_LATCH.Visu_Ret_Arr[13] := FALSE;
   TL_IDLE_LATCH.Visu_Ret_Arr[14] := FALSE;
   TL_IDLE_LATCH.Visu_Ret_Arr[15] := FALSE;
   TL_IDLE_LATCH.BLK_Move_Ret := 0;
   TL_IDLE_LATCH.Enable := FALSE;
   TL_IDLE_LATCH.Adv_End := FALSE;
   TL_IDLE_LATCH.Ret_End := FALSE;
   TL_IDLE_PIN.Enable_Aux := FALSE;
   TL_IDLE_PIN.Adv_Amount := 0;
   TL_IDLE_PIN.Ret_Amount := 0;
   TL_IDLE_PIN.LS_Adv1 := FALSE;
   TL_IDLE_PIN.LS_Ret1 := FALSE;
   TL_IDLE_PIN.LS_Adv2 := FALSE;
   TL_IDLE_PIN.LS_Ret2 := FALSE;
   TL_IDLE_PIN.LS_Adv3 := FALSE;
   TL_IDLE_PIN.LS_Ret3 := FALSE;
   TL_IDLE_PIN.LS_Adv4 := FALSE;
   TL_IDLE_PIN.LS_Ret4 := FALSE;
   TL_IDLE_PIN.SOL_Adv := FALSE;
   TL_IDLE_PIN.SOL_Ret := FALSE;
   TL_IDLE_PIN.M_Ready := FALSE;
   TL_IDLE_PIN.T_CHK1 := T#0MS;
   TL_IDLE_PIN.T_CHK2 := T#0MS;
   TL_IDLE_PIN.PB_Lamp_CHK := FALSE;
   TL_IDLE_PIN.PB_Error_Rst := FALSE;
   TL_IDLE_PIN.M_FLICK := FALSE;
   TL_IDLE_PIN.M_Adv_Err := FALSE;
   TL_IDLE_PIN.M_Ret_Err := FALSE;
   TL_IDLE_PIN.LP_Adv := FALSE;
   TL_IDLE_PIN.LP_Ret := FALSE;
   TL_IDLE_PIN.Visu_Adv := W#16#0;
   TL_IDLE_PIN.Visu_Ret := W#16#0;
   TL_IDLE_PIN.Error_T1.IN := FALSE;
   TL_IDLE_PIN.Error_T1.PT := T#0MS;
   TL_IDLE_PIN.Error_T1.Q := FALSE;
   TL_IDLE_PIN.Error_T1.ET := T#0MS;
   TL_IDLE_PIN.Error_T1.STATE := B#16#0;
   TL_IDLE_PIN.Error_T1.STIME := T#0MS;
   TL_IDLE_PIN.Error_T1.ATIME := T#0MS;
   TL_IDLE_PIN.Error_T2.IN := FALSE;
   TL_IDLE_PIN.Error_T2.PT := T#0MS;
   TL_IDLE_PIN.Error_T2.Q := FALSE;
   TL_IDLE_PIN.Error_T2.ET := T#0MS;
   TL_IDLE_PIN.Error_T2.STATE := B#16#0;
   TL_IDLE_PIN.Error_T2.STIME := T#0MS;
   TL_IDLE_PIN.Error_T2.ATIME := T#0MS;
   TL_IDLE_PIN.CHK_Aux1 := FALSE;
   TL_IDLE_PIN.CHK_Aux2 := FALSE;
   TL_IDLE_PIN.Error_T1_DN := FALSE;
   TL_IDLE_PIN.Error_T2_DN := FALSE;
   TL_IDLE_PIN.Adv_Memo := FALSE;
   TL_IDLE_PIN.Visu_Adv_Arr[0] := FALSE;
   TL_IDLE_PIN.Visu_Adv_Arr[1] := FALSE;
   TL_IDLE_PIN.Visu_Adv_Arr[2] := FALSE;
   TL_IDLE_PIN.Visu_Adv_Arr[3] := FALSE;
   TL_IDLE_PIN.Visu_Adv_Arr[4] := FALSE;
   TL_IDLE_PIN.Visu_Adv_Arr[5] := FALSE;
   TL_IDLE_PIN.Visu_Adv_Arr[6] := FALSE;
   TL_IDLE_PIN.Visu_Adv_Arr[7] := FALSE;
   TL_IDLE_PIN.Visu_Adv_Arr[8] := FALSE;
   TL_IDLE_PIN.Visu_Adv_Arr[9] := FALSE;
   TL_IDLE_PIN.Visu_Adv_Arr[10] := FALSE;
   TL_IDLE_PIN.Visu_Adv_Arr[11] := FALSE;
   TL_IDLE_PIN.Visu_Adv_Arr[12] := FALSE;
   TL_IDLE_PIN.Visu_Adv_Arr[13] := FALSE;
   TL_IDLE_PIN.Visu_Adv_Arr[14] := FALSE;
   TL_IDLE_PIN.Visu_Adv_Arr[15] := FALSE;
   TL_IDLE_PIN.Visu_Ret_Arr[0] := FALSE;
   TL_IDLE_PIN.Visu_Ret_Arr[1] := FALSE;
   TL_IDLE_PIN.Visu_Ret_Arr[2] := FALSE;
   TL_IDLE_PIN.Visu_Ret_Arr[3] := FALSE;
   TL_IDLE_PIN.Visu_Ret_Arr[4] := FALSE;
   TL_IDLE_PIN.Visu_Ret_Arr[5] := FALSE;
   TL_IDLE_PIN.Visu_Ret_Arr[6] := FALSE;
   TL_IDLE_PIN.Visu_Ret_Arr[7] := FALSE;
   TL_IDLE_PIN.Visu_Ret_Arr[8] := FALSE;
   TL_IDLE_PIN.Visu_Ret_Arr[9] := FALSE;
   TL_IDLE_PIN.Visu_Ret_Arr[10] := FALSE;
   TL_IDLE_PIN.Visu_Ret_Arr[11] := FALSE;
   TL_IDLE_PIN.Visu_Ret_Arr[12] := FALSE;
   TL_IDLE_PIN.Visu_Ret_Arr[13] := FALSE;
   TL_IDLE_PIN.Visu_Ret_Arr[14] := FALSE;
   TL_IDLE_PIN.Visu_Ret_Arr[15] := FALSE;
   TL_IDLE_PIN.BLK_Move_Ret := 0;
   TL_IDLE_PIN.Enable := FALSE;
   TL_IDLE_PIN.Adv_End := FALSE;
   TL_IDLE_PIN.Ret_End := FALSE;
END_DATA_BLOCK

FUNCTION FC 111 : VOID
TITLE =
VERSION : 0.1

BEGIN
NETWORK
TITLE =WORK COMP'T
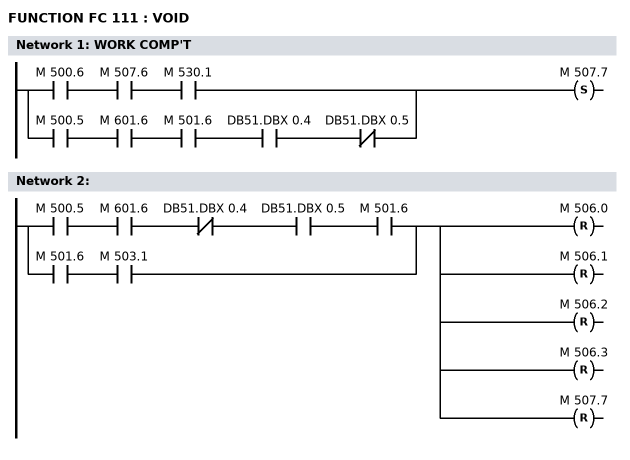

      A     M    500.6;
      A     M    507.6;
      A     M    530.1;
      O     ;
      A     M    500.5;
      A     M    601.6;
      A     M    501.6;
      A     DB51.DBX    0.4;
      AN    DB51.DBX    0.5;
      S     M    507.7;
NETWORK
TITLE =

      A     M    500.5;
      A     M    601.6;
      AN    DB51.DBX    0.4;
      A     DB51.DBX    0.5;
      A     M    501.6;
      O     ;
      A     M    501.6;
      A     M    503.1;
      R     M    506.0;
      R     M    506.1;
      R     M    506.2;
      R     M    506.3;
      R     M    507.7;
NETWORK
TITLE =GUN1,2,3,4 WELD'G COMP'T

      A     M    500.2;
      =     L      0.0;
      A     L      0.0;
      A     I     38.0;
      A     T     51;
      =     L      0.1;
      A     L      0.1;
      A     M    520.3;
      S     M    506.0;
      A     L      0.1;
      A     M    506.0;
      A     M    520.2;
      S     M    506.1;
      A     L      0.0;
      A     I     38.2;
      A     T     54;
      A     M    520.0;
      =     L      0.1;
      A     L      0.1;
      A     M    520.7;
      S     M    506.2;
      A     L      0.1;
      A     M    506.2;
      A     M    520.6;
      S     M    506.3;
NETWORK
TITLE =GUN1,2,3,4 WELD'G COMP'T, STN WORK COMP'T
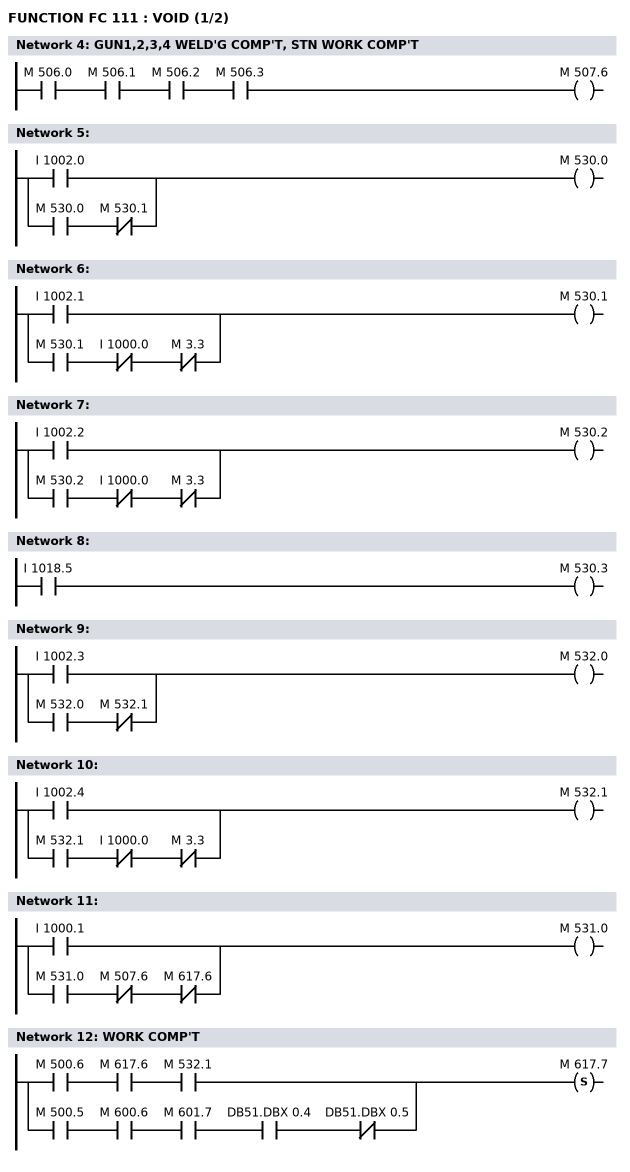

      A     M    506.0;
      A     M    506.1;
      A     M    506.2;
      A     M    506.3;
      =     M    507.6;
NETWORK
TITLE =

      O     I   1002.0;
      O     ;
      A     M    530.0;
      AN    M    530.1;
      =     M    530.0;
NETWORK
TITLE =

      O     I   1002.1;
      O     ;
      A     M    530.1;
      AN    I   1000.0;
      AN    M      3.3;
      =     M    530.1;
NETWORK
TITLE =

      O     I   1002.2;
      O     ;
      A     M    530.2;
      AN    I   1000.0;
      AN    M      3.3;
      =     M    530.2;
NETWORK
TITLE =

      A     I   1018.5;
      =     M    530.3;
NETWORK
TITLE =

      O     I   1002.3;
      O     ;
      A     M    532.0;
      AN    M    532.1;
      =     M    532.0;
NETWORK
TITLE =

      O     I   1002.4;
      O     ;
      A     M    532.1;
      AN    I   1000.0;
      AN    M      3.3;
      =     M    532.1;
NETWORK
TITLE =

      O     I   1000.1;
      O     ;
      A     M    531.0;
      AN    M    507.6;
      AN    M    617.6;
      =     M    531.0;
NETWORK
TITLE =WORK COMP'T

      A     M    500.6;
      A     M    617.6;
      A     M    532.1;
      O     ;
      A     M    500.5;
      A     M    600.6;
      A     M    601.7;
      A     DB51.DBX    0.4;
      AN    DB51.DBX    0.5;
      S     M    617.7;
NETWORK
TITLE =
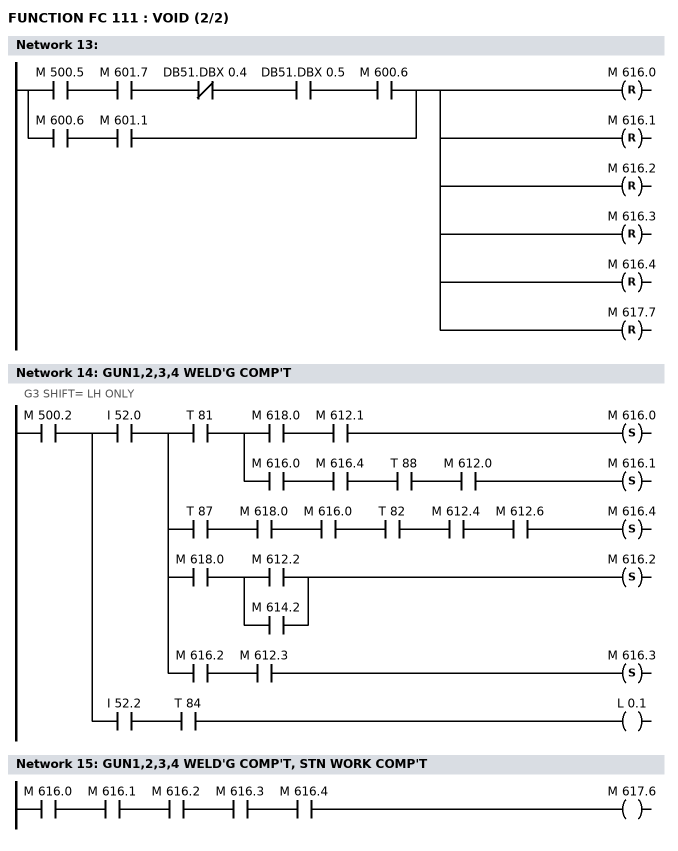

      A     M    500.5;
      A     M    601.7;
      AN    DB51.DBX    0.4;
      A     DB51.DBX    0.5;
      A     M    600.6;
      O     ;
      A     M    600.6;
      A     M    601.1;
      R     M    616.0;
      R     M    616.1;
      R     M    616.2;
      R     M    616.3;
      R     M    616.4;
      R     M    617.7;
NETWORK
TITLE =GUN1,2,3,4 WELD'G COMP'T
//G3 SHIFT= LH ONLY
      A     M    500.2;
      =     L      0.0;
      A     L      0.0;
      A     I     52.0;
      =     L      0.1;
      A     L      0.1;
      A     T     81;
      =     L      0.2;
      A     L      0.2;
      A     M    618.0;
      A     M    612.1;
      S     M    616.0;
      A     L      0.2;
      A     M    616.0;
      A     M    616.4;
      A     T     88;
      A     M    612.0;
      S     M    616.1;
      A     L      0.1;
      A     T     87;
      A     M    618.0;
      A     M    616.0;
      A     T     82;
      A     M    612.4;
      A     M    612.6;
      S     M    616.4;
      A     L      0.0;
      A     I     52.2;
      A     T     84;
      =     L      0.1;
      A     L      0.1;
      A     M    618.0;
      A(    ;
      O     M    612.2;
      O     M    614.2;
      )     ;
      S     M    616.2;
      A     L      0.1;
      A     M    616.2;
      A     M    612.3;
      S     M    616.3;
NETWORK
TITLE =GUN1,2,3,4 WELD'G COMP'T, STN WORK COMP'T

      A     M    616.0;
      A     M    616.1;
      A     M    616.2;
      A     M    616.3;
      A     M    616.4;
      =     M    617.6;
END_FUNCTION

FUNCTION_BLOCK FB 112
TITLE =
VERSION : 0.1

BEGIN
NETWORK
TITLE =

NETWORK
TITLE =LS ERROR
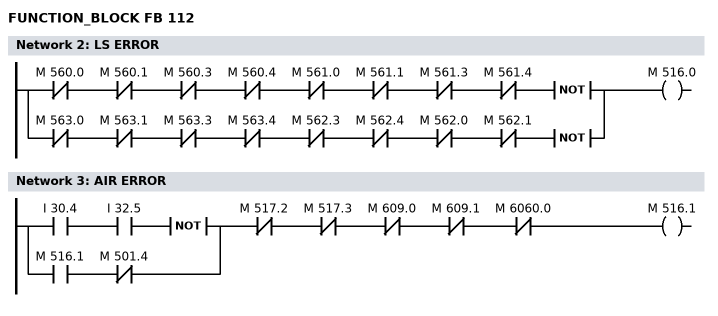

      AN    M    560.0;
      AN    M    560.1;
      AN    M    560.3;
      AN    M    560.4;
      AN    M    561.0;
      AN    M    561.1;
      AN    M    561.3;
      AN    M    561.4;
      NOT   ;
      O(    ;
      AN    M    563.0;
      AN    M    563.1;
      AN    M    563.3;
      AN    M    563.4;
      AN    M    562.3;
      AN    M    562.4;
      AN    M    562.0;
      AN    M    562.1;
      NOT   ;
      )     ;
      =     M    516.0;
NETWORK
TITLE =AIR ERROR

      A(    ;
      A     I     30.4;
      A     I     32.5;
      NOT   ;
      O     ;
      A     M    516.1;
      AN    M    501.4;
      )     ;
      AN    M    517.2;
      AN    M    517.3;
      AN    M    609.0;
      AN    M    609.1;
      AN    M   6060.0;
      =     M    516.1;
NETWORK
TITLE =WATER ERROR

      AN    OV;
      A(    ;
      O     I     35.7;
      O     ;
      A     M    516.2;
      AN    M    501.4;
      )     ;
      AN    M      3.3;
      AN    M    517.2;
      AN    M    517.3;
      AN    M    609.0;
      AN    M    609.1;
      AN    M   6060.0;
      =     M    516.2;
NETWORK
TITLE =MAT S/W ERROR
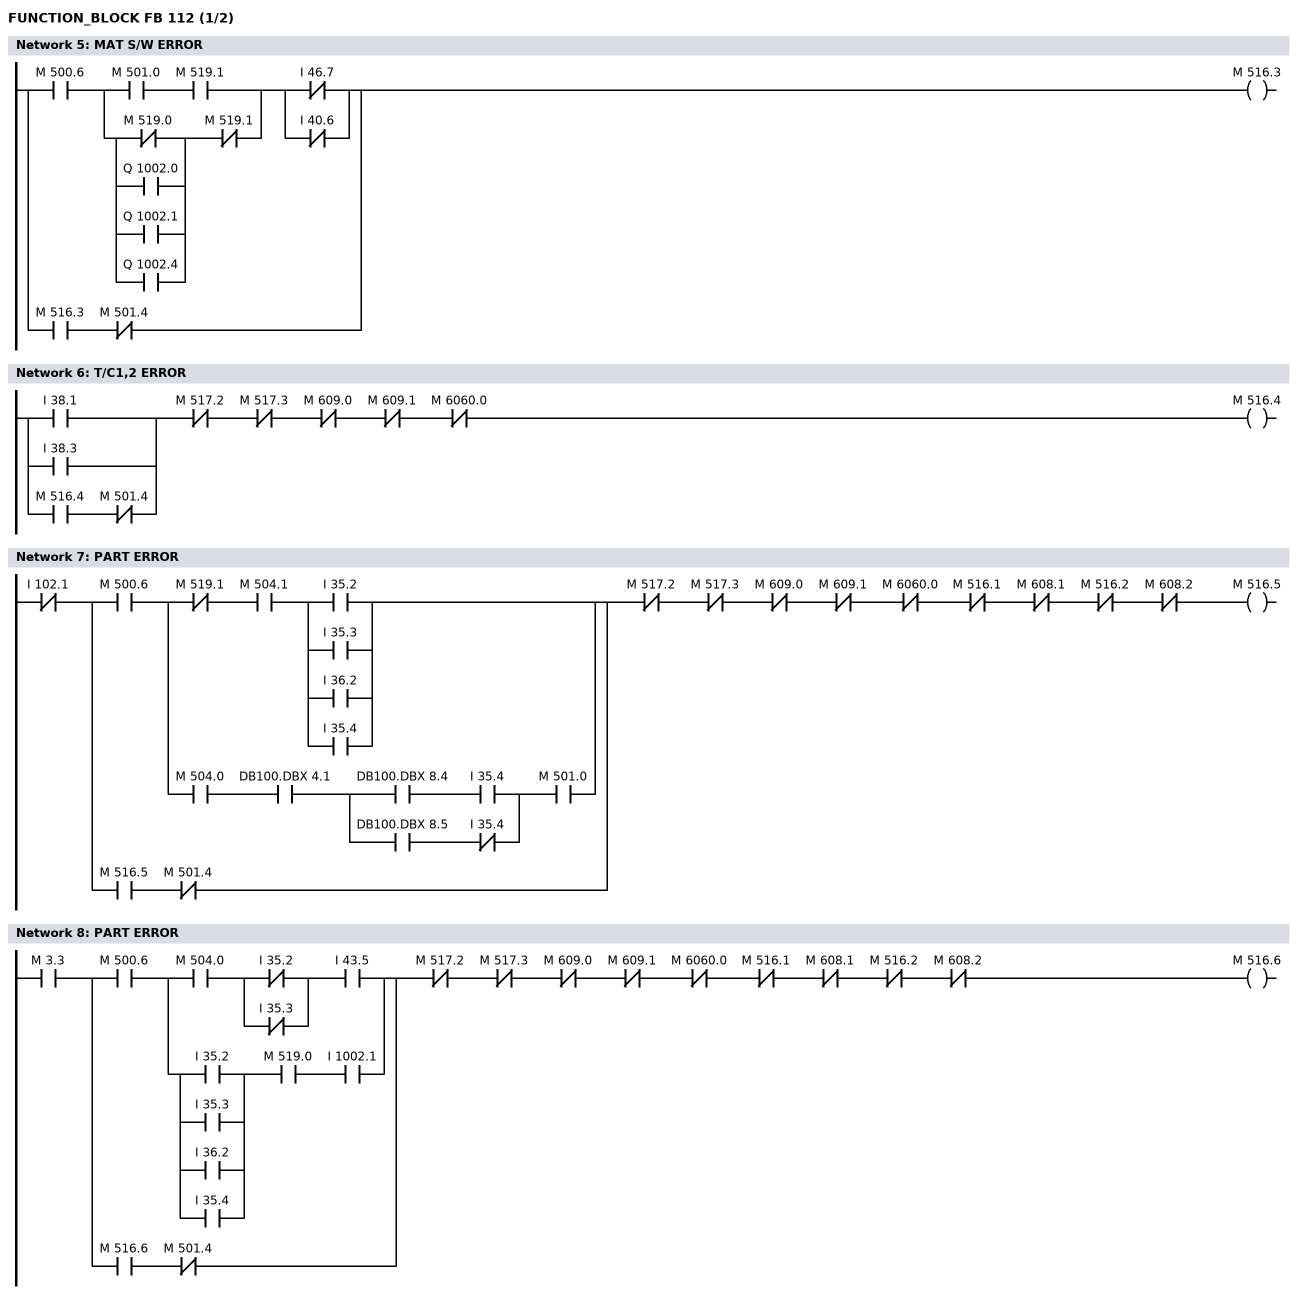

      A     M    500.6;
      A(    ;
      A     M    501.0;
      A     M    519.1;
      O     ;
      A(    ;
      ON    M    519.0;
      O     Q   1002.0;
      O     Q   1002.1;
      O     Q   1002.4;
      )     ;
      AN    M    519.1;
      )     ;
      A(    ;
      ON    I     46.7;
      ON    I     40.6;
      )     ;
      O     ;
      A     M    516.3;
      AN    M    501.4;
      =     M    516.3;
NETWORK
TITLE =T/C1,2 ERROR

      A(    ;
      O     I     38.1;
      O     I     38.3;
      O     ;
      A     M    516.4;
      AN    M    501.4;
      )     ;
      AN    M    517.2;
      AN    M    517.3;
      AN    M    609.0;
      AN    M    609.1;
      AN    M   6060.0;
      =     M    516.4;
NETWORK
TITLE =PART ERROR

      AN    I    102.1;
      A(    ;
      A     M    500.6;
      A(    ;
      AN    M    519.1;
      A     M    504.1;
      A(    ;
      O     I     35.2;
      O     I     35.3;
      O     I     36.2;
      O     I     35.4;
      )     ;
      O     ;
      A     M    504.0;
      A     DB100.DBX    4.1;
      A(    ;
      A     DB100.DBX    8.4;
      A     I     35.4;
      O     ;
      A     DB100.DBX    8.5;
      AN    I     35.4;
      )     ;
      A     M    501.0;
      )     ;
      O     ;
      A     M    516.5;
      AN    M    501.4;
      )     ;
      AN    M    517.2;
      AN    M    517.3;
      AN    M    609.0;
      AN    M    609.1;
      AN    M   6060.0;
      AN    M    516.1;
      AN    M    608.1;
      AN    M    516.2;
      AN    M    608.2;
      =     M    516.5;
NETWORK
TITLE =PART ERROR

      A     M      3.3;
      A(    ;
      A     M    500.6;
      A(    ;
      A     M    504.0;
      A(    ;
      ON    I     35.2;
      ON    I     35.3;
      )     ;
      A     I     43.5;
      O     ;
      A(    ;
      O     I     35.2;
      O     I     35.3;
      O     I     36.2;
      O     I     35.4;
      )     ;
      A     M    519.0;
      A     I   1002.1;
      )     ;
      O     ;
      A     M    516.6;
      AN    M    501.4;
      )     ;
      AN    M    517.2;
      AN    M    517.3;
      AN    M    609.0;
      AN    M    609.1;
      AN    M   6060.0;
      AN    M    516.1;
      AN    M    608.1;
      AN    M    516.2;
      AN    M    608.2;
      =     M    516.6;
NETWORK
TITLE =PART ERROR
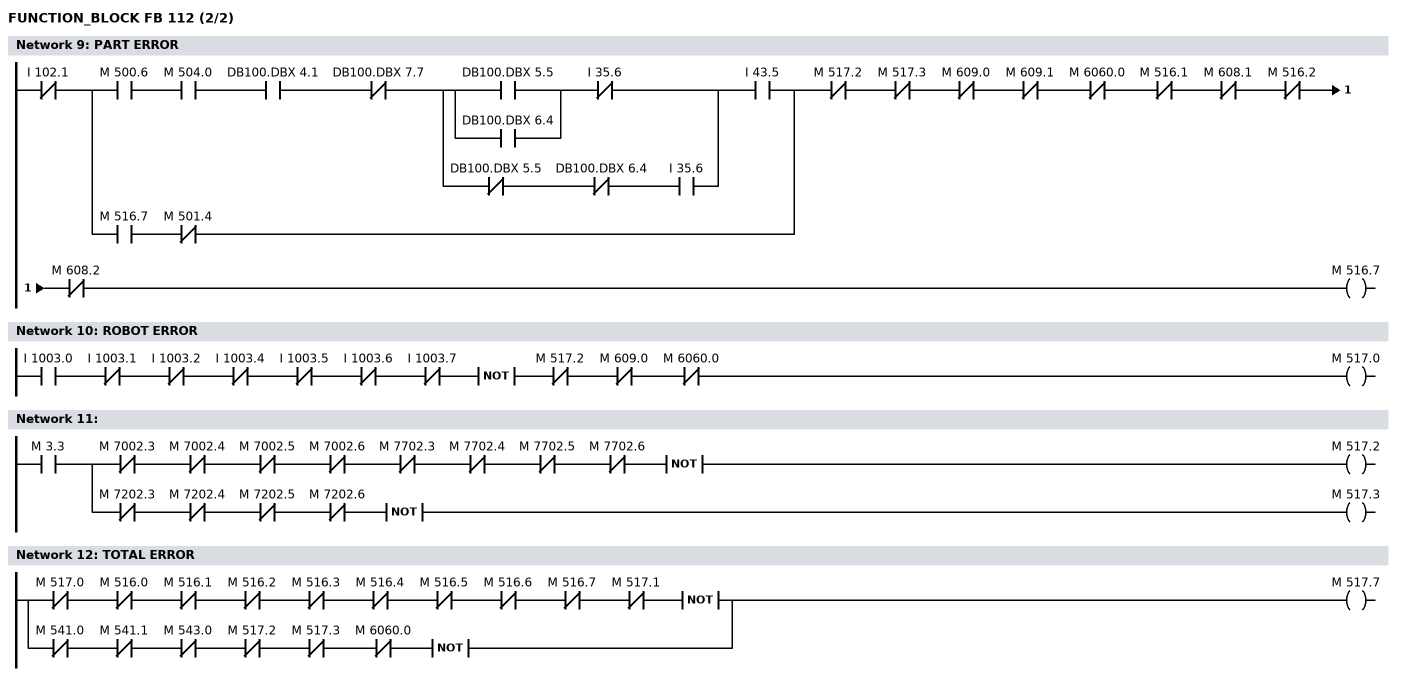

      AN    I    102.1;
      A(    ;
      A     M    500.6;
      A     M    504.0;
      A     DB100.DBX    4.1;
      AN    DB100.DBX    7.7;
      A(    ;
      A(    ;
      O     DB100.DBX    5.5;
      O     DB100.DBX    6.4;
      )     ;
      AN    I     35.6;
      O     ;
      AN    DB100.DBX    5.5;
      AN    DB100.DBX    6.4;
      A     I     35.6;
      )     ;
      A     I     43.5;
      O     ;
      A     M    516.7;
      AN    M    501.4;
      )     ;
      AN    M    517.2;
      AN    M    517.3;
      AN    M    609.0;
      AN    M    609.1;
      AN    M   6060.0;
      AN    M    516.1;
      AN    M    608.1;
      AN    M    516.2;
      AN    M    608.2;
      =     M    516.7;
NETWORK
TITLE =ROBOT ERROR

      A     I   1003.0;
      AN    I   1003.1;
      AN    I   1003.2;
      AN    I   1003.4;
      AN    I   1003.5;
      AN    I   1003.6;
      AN    I   1003.7;
      NOT   ;
      AN    M    517.2;
      AN    M    609.0;
      AN    M   6060.0;
      =     M    517.0;
NETWORK
TITLE =

      A     M      3.3;
      =     L      0.0;
      A     L      0.0;
      AN    M   7002.3;
      AN    M   7002.4;
      AN    M   7002.5;
      AN    M   7002.6;
      AN    M   7702.3;
      AN    M   7702.4;
      AN    M   7702.5;
      AN    M   7702.6;
      NOT   ;
      =     M    517.2;
      A     L      0.0;
      AN    M   7202.3;
      AN    M   7202.4;
      AN    M   7202.5;
      AN    M   7202.6;
      NOT   ;
      =     M    517.3;
NETWORK
TITLE =TOTAL ERROR

      AN    M    517.0;
      AN    M    516.0;
      AN    M    516.1;
      AN    M    516.2;
      AN    M    516.3;
      AN    M    516.4;
      AN    M    516.5;
      AN    M    516.6;
      AN    M    516.7;
      AN    M    517.1;
      NOT   ;
      O(    ;
      AN    M    541.0;
      AN    M    541.1;
      AN    M    543.0;
      AN    M    517.2;
      AN    M    517.3;
      AN    M   6060.0;
      NOT   ;
      )     ;
      =     M    517.7;
NETWORK
TITLE =

NETWORK
TITLE =

      AN    OV;
      A(    ;
      A     M    505.1;
      A     I   1002.7;
      A     I   1018.4;
      AN    I   1002.2;
      A(    ;
      O     I     32.2;
      O     I     32.3;
      O     I     33.6;
      O     I     33.7;
      )     ;
      O     ;
      A     M    541.0;
      AN    M    501.4;
      )     ;
      AN    M    517.2;
      AN    M    517.3;
      AN    M    609.0;
      AN    M    609.1;
      AN    M   6060.0;
      AN    M    516.1;
      AN    M    608.1;
      AN    M    516.2;
      AN    M    608.2;
      =     M    541.0;
NETWORK
TITLE =

      AN    OV;
      =     L      0.0;
      A     L      0.0;
      A     M    505.0;
      A     I   1002.7;
      A     M    531.2;
      A(    ;
      A     DB100.DBX   44.1;
      A(    ;
      ON    I     32.2;
      O     ;
      A(    ;
      ON    I     32.3;
      O     I     32.6;
      )     ;
      A     DB100.DBX   48.4;
      AN    DB100.DBX   47.7;
      O     ;
      A(    ;
      O     I     32.3;
      O     I     32.6;
      )     ;
      A     DB100.DBX   48.5;
      AN    DB100.DBX   47.7;
      O     ;
      AN    I     32.6;
      A     DB100.DBX   47.7;
      )     ;
      O     ;
      A     DB100.DBX   44.0;
      A(    ;
      ON    I     33.6;
      ON    I     33.7;
      )     ;
      )     ;
      =     L      0.1;
      A     L      0.1;
      A     T     70;
      S     M    541.1;
      A     L      0.1;
      AN    M    517.2;
      AN    M    517.3;
      AN    M    609.0;
      AN    M    609.1;
      AN    M   6060.0;
      AN    M    516.1;
      AN    M    608.1;
      AN    M    516.2;
      AN    M    608.2;
      L     S5T#4S500MS;
      SD    T     70;
      A     L      0.0;
      A     M    541.1;
      A     M    501.4;
      A(    ;
      A     DB100.DBX   44.1;
      A     I     32.2;
      A(    ;
      AN    I     32.6;
      AN    DB100.DBX   47.7;
      A(    ;
      A     I     32.3;
      A     DB100.DBX   48.4;
      O     ;
      AN    I     32.3;
      A     DB100.DBX   48.5;
      )     ;
      O     ;
      A     I     32.6;
      A     DB100.DBX   47.7;
      )     ;
      O     ;
      A     DB100.DBX   44.0;
      A     I     33.6;
      A     I     33.7;
      O     ;
      AN    DB100.DBX   44.0;
      AN    I     33.6;
      AN    I     33.7;
      )     ;
      R     M    541.1;
      A     L      0.0;
      A(    ;
      O     I   1002.2;
      O     M    531.2;
      )     ;
      AN    T     30;
      =     M    531.2;
      L     S5T#5S;
      SD    T     30;
NETWORK
TITLE =
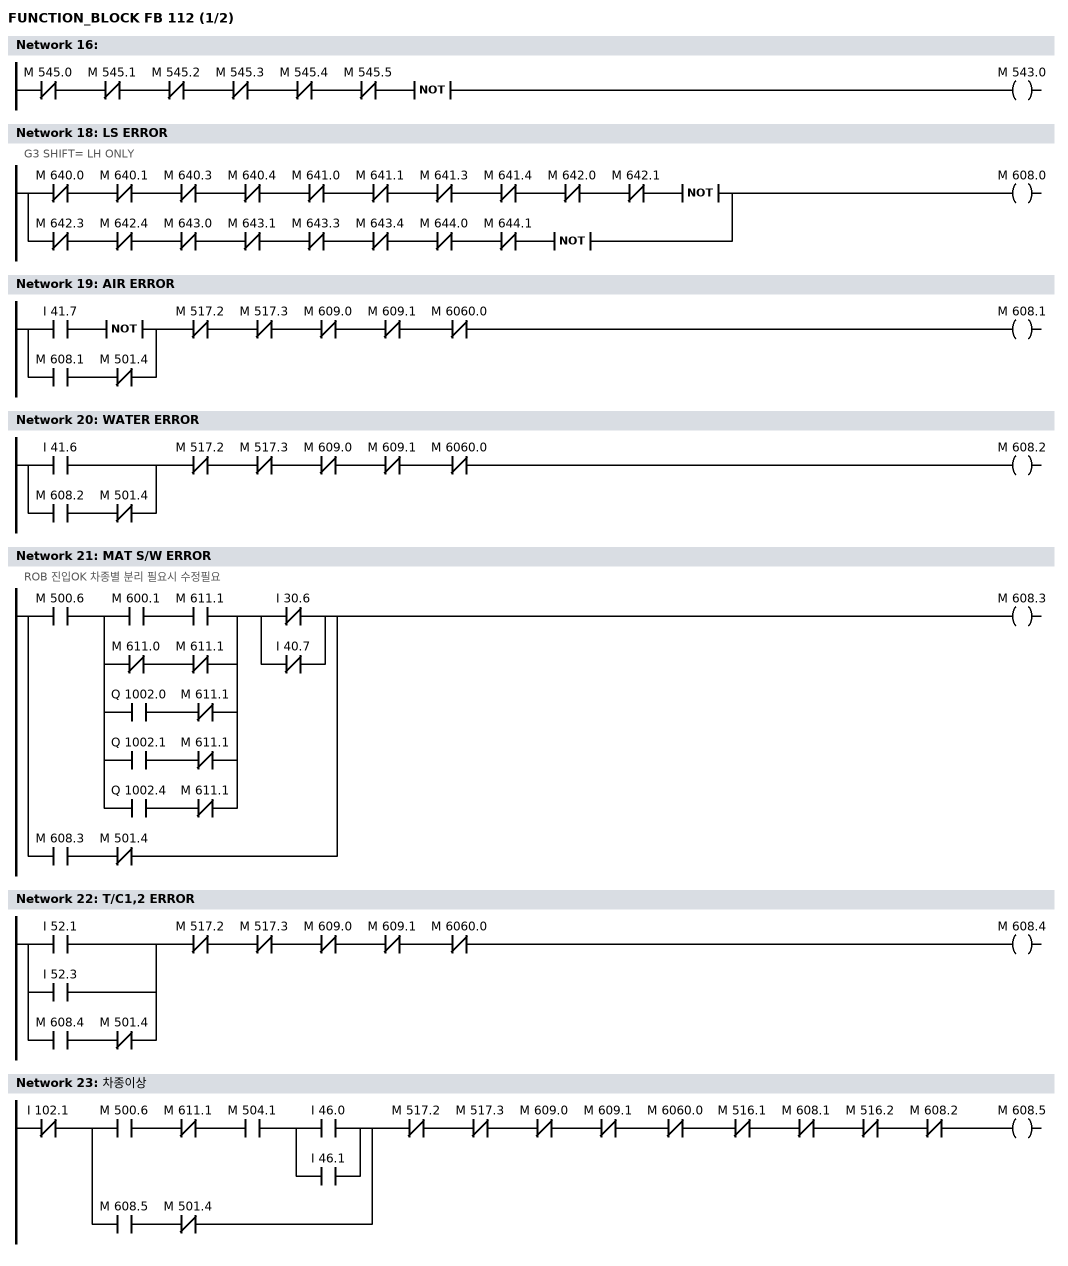

      AN    M    545.0;
      AN    M    545.1;
      AN    M    545.2;
      AN    M    545.3;
      AN    M    545.4;
      AN    M    545.5;
      NOT   ;
      =     M    543.0;
NETWORK
TITLE =

NETWORK
TITLE =LS ERROR
//G3 SHIFT= LH ONLY
      AN    M    640.0;
      AN    M    640.1;
      AN    M    640.3;
      AN    M    640.4;
      AN    M    641.0;
      AN    M    641.1;
      AN    M    641.3;
      AN    M    641.4;
      AN    M    642.0;
      AN    M    642.1;
      NOT   ;
      O(    ;
      AN    M    642.3;
      AN    M    642.4;
      AN    M    643.0;
      AN    M    643.1;
      AN    M    643.3;
      AN    M    643.4;
      AN    M    644.0;
      AN    M    644.1;
      NOT   ;
      )     ;
      =     M    608.0;
NETWORK
TITLE =AIR ERROR

      A(    ;
      A     I     41.7;
      NOT   ;
      O     ;
      A     M    608.1;
      AN    M    501.4;
      )     ;
      AN    M    517.2;
      AN    M    517.3;
      AN    M    609.0;
      AN    M    609.1;
      AN    M   6060.0;
      =     M    608.1;
NETWORK
TITLE =WATER ERROR

      A(    ;
      O     I     41.6;
      O     ;
      A     M    608.2;
      AN    M    501.4;
      )     ;
      AN    M    517.2;
      AN    M    517.3;
      AN    M    609.0;
      AN    M    609.1;
      AN    M   6060.0;
      =     M    608.2;
NETWORK
TITLE =MAT S/W ERROR
//ROB 진입OK 차종별 분리 필요시 수정필요
      A     M    500.6;
      A(    ;
      A     M    600.1;
      A     M    611.1;
      O     ;
      AN    M    611.0;
      AN    M    611.1;
      O     ;
      A     Q   1002.0;
      AN    M    611.1;
      O     ;
      A     Q   1002.1;
      AN    M    611.1;
      O     ;
      A     Q   1002.4;
      AN    M    611.1;
      )     ;
      A(    ;
      ON    I     30.6;
      ON    I     40.7;
      )     ;
      O     ;
      A     M    608.3;
      AN    M    501.4;
      =     M    608.3;
NETWORK
TITLE =T/C1,2 ERROR

      A(    ;
      O     I     52.1;
      O     I     52.3;
      O     ;
      A     M    608.4;
      AN    M    501.4;
      )     ;
      AN    M    517.2;
      AN    M    517.3;
      AN    M    609.0;
      AN    M    609.1;
      AN    M   6060.0;
      =     M    608.4;
NETWORK
TITLE =차종이상

      AN    I    102.1;
      A(    ;
      A     M    500.6;
      AN    M    611.1;
      A     M    504.1;
      A(    ;
      O     I     46.0;
      O     I     46.1;
      )     ;
      O     ;
      A     M    608.5;
      AN    M    501.4;
      )     ;
      AN    M    517.2;
      AN    M    517.3;
      AN    M    609.0;
      AN    M    609.1;
      AN    M   6060.0;
      AN    M    516.1;
      AN    M    608.1;
      AN    M    516.2;
      AN    M    608.2;
      =     M    608.5;
NETWORK
TITLE =PART ERROR
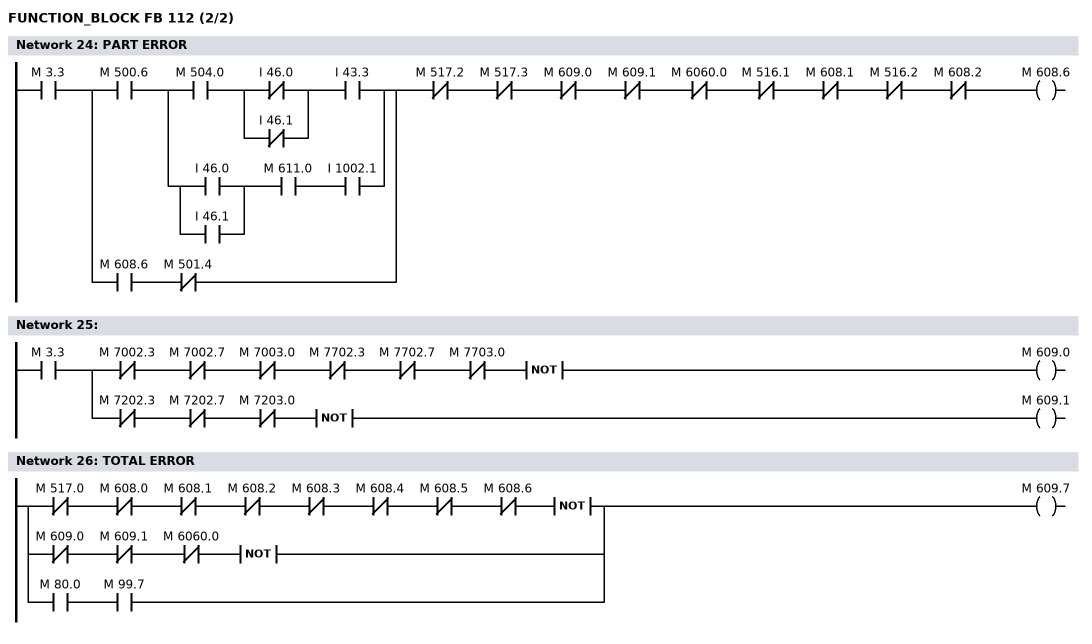

      A     M      3.3;
      A(    ;
      A     M    500.6;
      A(    ;
      A     M    504.0;
      A(    ;
      ON    I     46.0;
      ON    I     46.1;
      )     ;
      A     I     43.3;
      O     ;
      A(    ;
      O     I     46.0;
      O     I     46.1;
      )     ;
      A     M    611.0;
      A     I   1002.1;
      )     ;
      O     ;
      A     M    608.6;
      AN    M    501.4;
      )     ;
      AN    M    517.2;
      AN    M    517.3;
      AN    M    609.0;
      AN    M    609.1;
      AN    M   6060.0;
      AN    M    516.1;
      AN    M    608.1;
      AN    M    516.2;
      AN    M    608.2;
      =     M    608.6;
NETWORK
TITLE =

      A     M      3.3;
      =     L      0.0;
      A     L      0.0;
      AN    M   7002.3;
      AN    M   7002.7;
      AN    M   7003.0;
      AN    M   7702.3;
      AN    M   7702.7;
      AN    M   7703.0;
      NOT   ;
      =     M    609.0;
      A     L      0.0;
      AN    M   7202.3;
      AN    M   7202.7;
      AN    M   7203.0;
      NOT   ;
      =     M    609.1;
NETWORK
TITLE =TOTAL ERROR

      AN    M    517.0;
      AN    M    608.0;
      AN    M    608.1;
      AN    M    608.2;
      AN    M    608.3;
      AN    M    608.4;
      AN    M    608.5;
      AN    M    608.6;
      NOT   ;
      O(    ;
      AN    M    609.0;
      AN    M    609.1;
      AN    M   6060.0;
      NOT   ;
      )     ;
      O     ;
      A     M     80.0;
      A     M     99.7;
      =     M    609.7;
END_FUNCTION_BLOCK

DATA_BLOCK DB 112
TITLE =
VERSION : 0.0

 FB 112
BEGIN
END_DATA_BLOCK

FUNCTION FC 112 : VOID
TITLE =
VERSION : 0.1

BEGIN
NETWORK
TITLE =LM KEY 공정

NETWORK
TITLE =PIN ADV/REV END
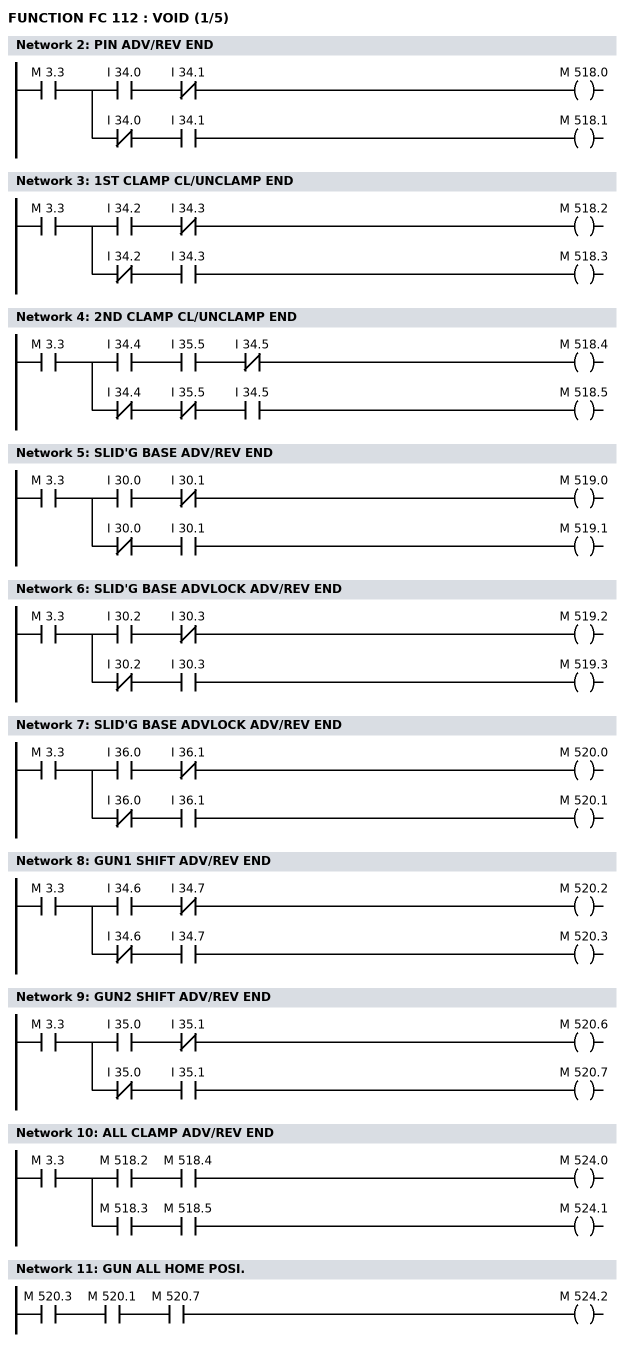

      A     M      3.3;
      =     L      0.0;
      A     L      0.0;
      A     I     34.0;
      AN    I     34.1;
      =     M    518.0;
      A     L      0.0;
      AN    I     34.0;
      A     I     34.1;
      =     M    518.1;
NETWORK
TITLE =1ST CLAMP CL/UNCLAMP END

      A     M      3.3;
      =     L      0.0;
      A     L      0.0;
      A     I     34.2;
      AN    I     34.3;
      =     M    518.2;
      A     L      0.0;
      AN    I     34.2;
      A     I     34.3;
      =     M    518.3;
NETWORK
TITLE =2ND CLAMP CL/UNCLAMP END

      A     M      3.3;
      =     L      0.0;
      A     L      0.0;
      A     I     34.4;
      A     I     35.5;
      AN    I     34.5;
      =     M    518.4;
      A     L      0.0;
      AN    I     34.4;
      AN    I     35.5;
      A     I     34.5;
      =     M    518.5;
NETWORK
TITLE =SLID'G BASE ADV/REV END

      A     M      3.3;
      =     L      0.0;
      A     L      0.0;
      A     I     30.0;
      AN    I     30.1;
      =     M    519.0;
      A     L      0.0;
      AN    I     30.0;
      A     I     30.1;
      =     M    519.1;
NETWORK
TITLE =SLID'G BASE ADVLOCK ADV/REV END

      A     M      3.3;
      =     L      0.0;
      A     L      0.0;
      A     I     30.2;
      AN    I     30.3;
      =     M    519.2;
      A     L      0.0;
      AN    I     30.2;
      A     I     30.3;
      =     M    519.3;
NETWORK
TITLE =SLID'G BASE ADVLOCK ADV/REV END

      A     M      3.3;
      =     L      0.0;
      A     L      0.0;
      A     I     36.0;
      AN    I     36.1;
      =     M    520.0;
      A     L      0.0;
      AN    I     36.0;
      A     I     36.1;
      =     M    520.1;
NETWORK
TITLE =GUN1 SHIFT ADV/REV END

      A     M      3.3;
      =     L      0.0;
      A     L      0.0;
      A     I     34.6;
      AN    I     34.7;
      =     M    520.2;
      A     L      0.0;
      AN    I     34.6;
      A     I     34.7;
      =     M    520.3;
NETWORK
TITLE =GUN2 SHIFT ADV/REV END

      A     M      3.3;
      =     L      0.0;
      A     L      0.0;
      A     I     35.0;
      AN    I     35.1;
      =     M    520.6;
      A     L      0.0;
      AN    I     35.0;
      A     I     35.1;
      =     M    520.7;
NETWORK
TITLE =ALL CLAMP ADV/REV END

      A     M      3.3;
      =     L      0.0;
      A     L      0.0;
      A     M    518.2;
      A     M    518.4;
      =     M    524.0;
      A     L      0.0;
      A     M    518.3;
      A     M    518.5;
      =     M    524.1;
NETWORK
TITLE =GUN ALL HOME POSI.

      A     M    520.3;
      A     M    520.1;
      A     M    520.7;
      =     M    524.2;
NETWORK
TITLE =PIN ADV
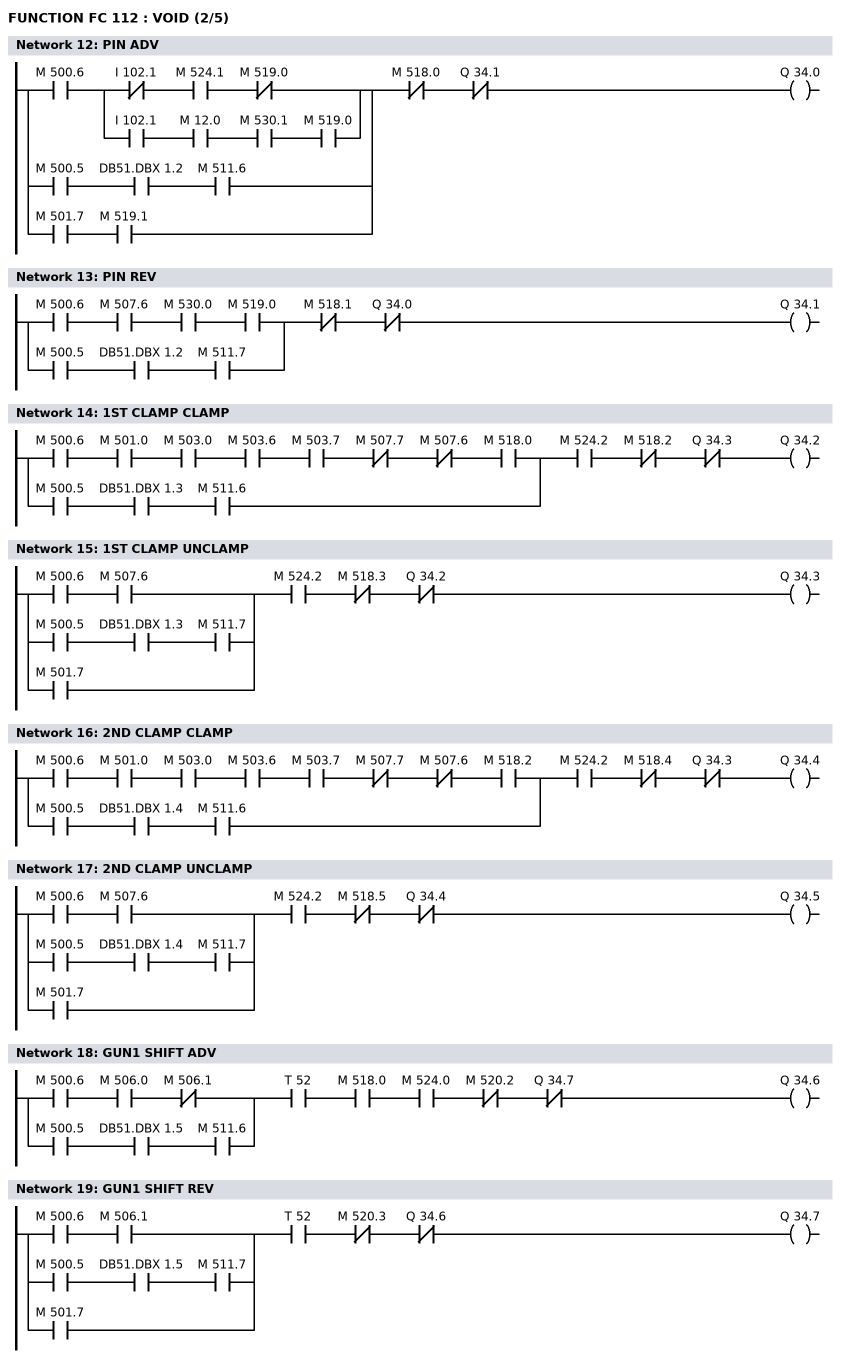

      A(    ;
      A     M    500.6;
      A(    ;
      AN    I    102.1;
      A     M    524.1;
      AN    M    519.0;
      O     ;
      A     I    102.1;
      A     M     12.0;
      A     M    530.1;
      A     M    519.0;
      )     ;
      O     ;
      A     M    500.5;
      A     DB51.DBX    1.2;
      A     M    511.6;
      O     ;
      A     M    501.7;
      A     M    519.1;
      )     ;
      AN    M    518.0;
      AN    Q     34.1;
      =     Q     34.0;
NETWORK
TITLE =PIN REV

      A(    ;
      A     M    500.6;
      A     M    507.6;
      A     M    530.0;
      A     M    519.0;
      O     ;
      A     M    500.5;
      A     DB51.DBX    1.2;
      A     M    511.7;
      )     ;
      AN    M    518.1;
      AN    Q     34.0;
      =     Q     34.1;
NETWORK
TITLE =1ST CLAMP CLAMP

      A(    ;
      A     M    500.6;
      A     M    501.0;
      A     M    503.0;
      A     M    503.6;
      A     M    503.7;
      AN    M    507.7;
      AN    M    507.6;
      A     M    518.0;
      O     ;
      A     M    500.5;
      A     DB51.DBX    1.3;
      A     M    511.6;
      )     ;
      A     M    524.2;
      AN    M    518.2;
      AN    Q     34.3;
      =     Q     34.2;
NETWORK
TITLE =1ST CLAMP UNCLAMP

      A(    ;
      A     M    500.6;
      A     M    507.6;
      O     ;
      A     M    500.5;
      A     DB51.DBX    1.3;
      A     M    511.7;
      O     M    501.7;
      )     ;
      A     M    524.2;
      AN    M    518.3;
      AN    Q     34.2;
      =     Q     34.3;
NETWORK
TITLE =2ND CLAMP CLAMP

      A(    ;
      A     M    500.6;
      A     M    501.0;
      A     M    503.0;
      A     M    503.6;
      A     M    503.7;
      AN    M    507.7;
      AN    M    507.6;
      A     M    518.2;
      O     ;
      A     M    500.5;
      A     DB51.DBX    1.4;
      A     M    511.6;
      )     ;
      A     M    524.2;
      AN    M    518.4;
      AN    Q     34.3;
      =     Q     34.4;
NETWORK
TITLE =2ND CLAMP UNCLAMP

      A(    ;
      A     M    500.6;
      A     M    507.6;
      O     ;
      A     M    500.5;
      A     DB51.DBX    1.4;
      A     M    511.7;
      O     M    501.7;
      )     ;
      A     M    524.2;
      AN    M    518.5;
      AN    Q     34.4;
      =     Q     34.5;
NETWORK
TITLE =GUN1 SHIFT ADV

      A(    ;
      A     M    500.6;
      A     M    506.0;
      AN    M    506.1;
      O     ;
      A     M    500.5;
      A     DB51.DBX    1.5;
      A     M    511.6;
      )     ;
      A     T     52;
      A     M    518.0;
      A     M    524.0;
      AN    M    520.2;
      AN    Q     34.7;
      =     Q     34.6;
NETWORK
TITLE =GUN1 SHIFT REV

      A(    ;
      A     M    500.6;
      A     M    506.1;
      O     ;
      A     M    500.5;
      A     DB51.DBX    1.5;
      A     M    511.7;
      O     M    501.7;
      )     ;
      A     T     52;
      AN    M    520.3;
      AN    Q     34.6;
      =     Q     34.7;
NETWORK
TITLE =1ST CLAMP CLAMP
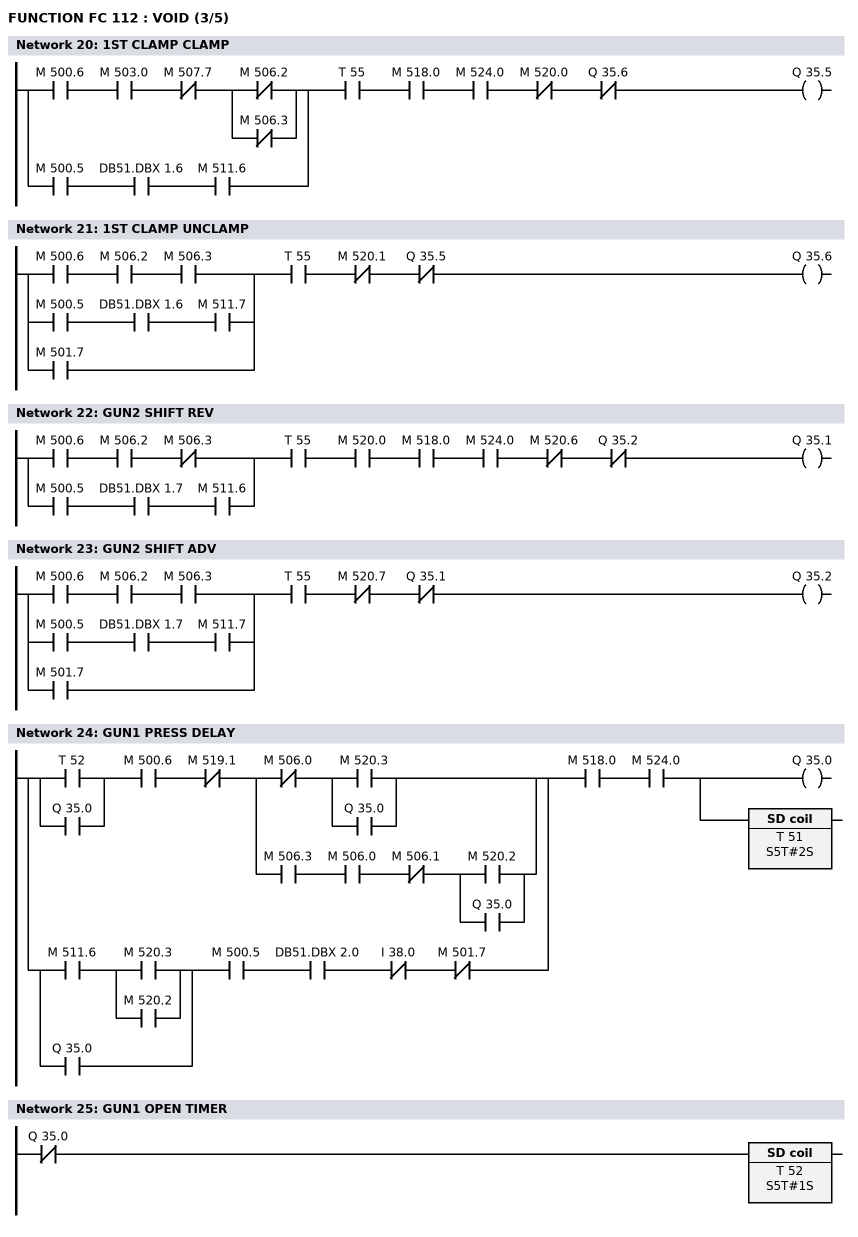

      A(    ;
      A     M    500.6;
      A     M    503.0;
      AN    M    507.7;
      A(    ;
      ON    M    506.2;
      ON    M    506.3;
      )     ;
      O     ;
      A     M    500.5;
      A     DB51.DBX    1.6;
      A     M    511.6;
      )     ;
      A     T     55;
      A     M    518.0;
      A     M    524.0;
      AN    M    520.0;
      AN    Q     35.6;
      =     Q     35.5;
NETWORK
TITLE =1ST CLAMP UNCLAMP

      A(    ;
      A     M    500.6;
      A     M    506.2;
      A     M    506.3;
      O     ;
      A     M    500.5;
      A     DB51.DBX    1.6;
      A     M    511.7;
      O     M    501.7;
      )     ;
      A     T     55;
      AN    M    520.1;
      AN    Q     35.5;
      =     Q     35.6;
NETWORK
TITLE =GUN2 SHIFT REV

      A(    ;
      A     M    500.6;
      A     M    506.2;
      AN    M    506.3;
      O     ;
      A     M    500.5;
      A     DB51.DBX    1.7;
      A     M    511.6;
      )     ;
      A     T     55;
      A     M    520.0;
      A     M    518.0;
      A     M    524.0;
      AN    M    520.6;
      AN    Q     35.2;
      =     Q     35.1;
NETWORK
TITLE =GUN2 SHIFT ADV

      A(    ;
      A     M    500.6;
      A     M    506.2;
      A     M    506.3;
      O     ;
      A     M    500.5;
      A     DB51.DBX    1.7;
      A     M    511.7;
      O     M    501.7;
      )     ;
      A     T     55;
      AN    M    520.7;
      AN    Q     35.1;
      =     Q     35.2;
NETWORK
TITLE =GUN1 PRESS DELAY

      A(    ;
      A(    ;
      O     T     52;
      O     Q     35.0;
      )     ;
      A     M    500.6;
      AN    M    519.1;
      A(    ;
      AN    M    506.0;
      A(    ;
      O     M    520.3;
      O     Q     35.0;
      )     ;
      O     ;
      A     M    506.3;
      A     M    506.0;
      AN    M    506.1;
      A(    ;
      O     M    520.2;
      O     Q     35.0;
      )     ;
      )     ;
      O     ;
      A(    ;
      A     M    511.6;
      A(    ;
      O     M    520.3;
      O     M    520.2;
      )     ;
      O     Q     35.0;
      )     ;
      A     M    500.5;
      A     DB51.DBX    2.0;
      AN    I     38.0;
      AN    M    501.7;
      )     ;
      A     M    518.0;
      A     M    524.0;
      =     Q     35.0;
      L     S5T#2S;
      SD    T     51;
NETWORK
TITLE =GUN1 OPEN TIMER

      AN    Q     35.0;
      L     S5T#1S;
      SD    T     52;
NETWORK
TITLE =GUN2 PRESS DELAY
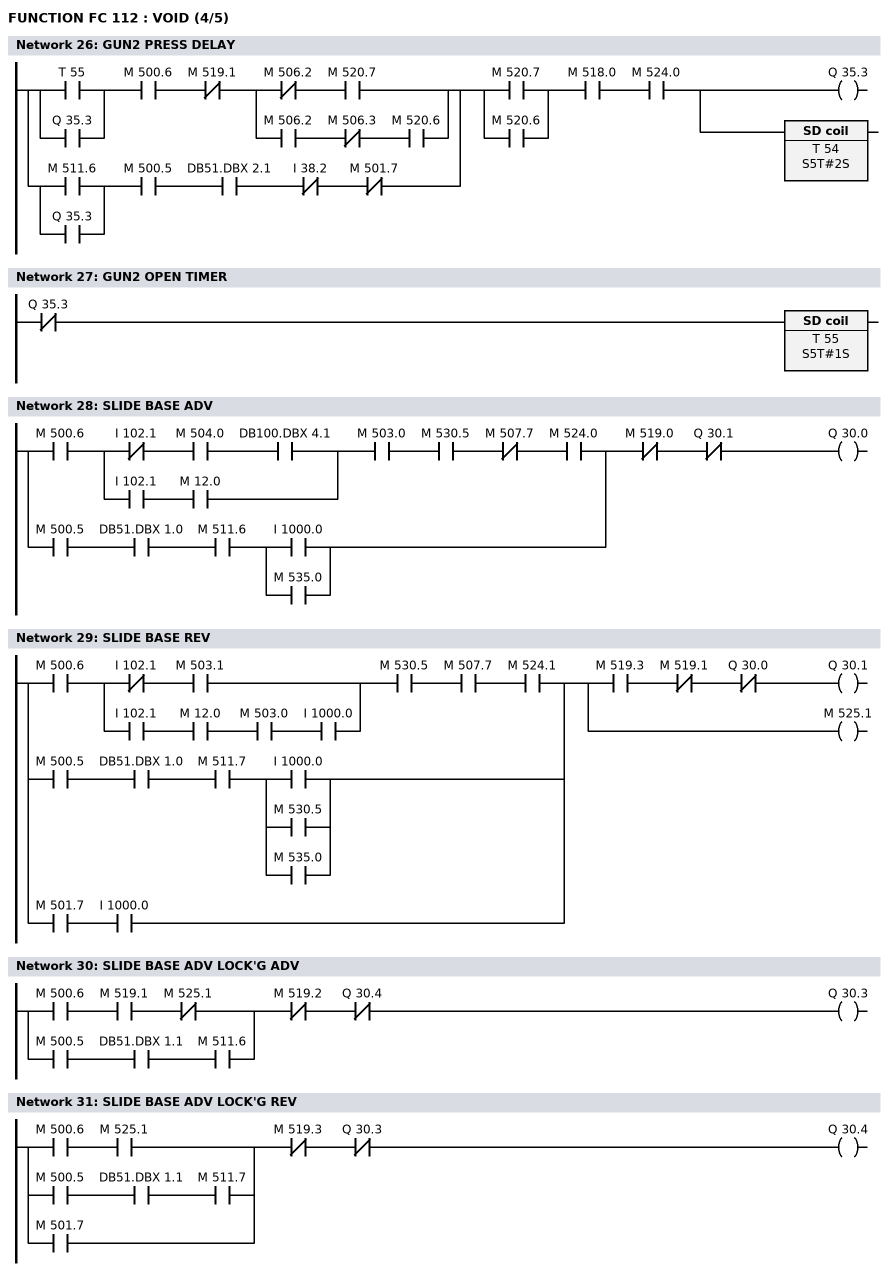

      A(    ;
      A(    ;
      O     T     55;
      O     Q     35.3;
      )     ;
      A     M    500.6;
      AN    M    519.1;
      A(    ;
      AN    M    506.2;
      A     M    520.7;
      O     ;
      A     M    506.2;
      AN    M    506.3;
      A     M    520.6;
      )     ;
      O     ;
      A(    ;
      O     M    511.6;
      O     Q     35.3;
      )     ;
      A     M    500.5;
      A     DB51.DBX    2.1;
      AN    I     38.2;
      AN    M    501.7;
      )     ;
      A(    ;
      O     M    520.7;
      O     M    520.6;
      )     ;
      A     M    518.0;
      A     M    524.0;
      =     Q     35.3;
      L     S5T#2S;
      SD    T     54;
NETWORK
TITLE =GUN2 OPEN TIMER

      AN    Q     35.3;
      L     S5T#1S;
      SD    T     55;
NETWORK
TITLE =SLIDE BASE ADV

      A(    ;
      A     M    500.6;
      A(    ;
      AN    I    102.1;
      A     M    504.0;
      A     DB100.DBX    4.1;
      O     ;
      A     I    102.1;
      A     M     12.0;
      )     ;
      A     M    503.0;
      A     M    530.5;
      AN    M    507.7;
      A     M    524.0;
      O     ;
      A     M    500.5;
      A     DB51.DBX    1.0;
      A     M    511.6;
      A(    ;
      O     I   1000.0;
      O     M    535.0;
      )     ;
      )     ;
      AN    M    519.0;
      AN    Q     30.1;
      =     Q     30.0;
NETWORK
TITLE =SLIDE BASE REV

      A     M    500.6;
      A(    ;
      AN    I    102.1;
      A     M    503.1;
      O     ;
      A     I    102.1;
      A     M     12.0;
      A     M    503.0;
      A     I   1000.0;
      )     ;
      A     M    530.5;
      A     M    507.7;
      A     M    524.1;
      O     ;
      A     M    500.5;
      A     DB51.DBX    1.0;
      A     M    511.7;
      A(    ;
      O     I   1000.0;
      O     M    530.5;
      O     M    535.0;
      )     ;
      O     ;
      A     M    501.7;
      A     I   1000.0;
      =     L      0.0;
      A     L      0.0;
      A     M    519.3;
      AN    M    519.1;
      AN    Q     30.0;
      =     Q     30.1;
      A     L      0.0;
      BLD   102;
      =     M    525.1;
NETWORK
TITLE =SLIDE BASE ADV LOCK'G ADV

      A(    ;
      A     M    500.6;
      A     M    519.1;
      AN    M    525.1;
      O     ;
      A     M    500.5;
      A     DB51.DBX    1.1;
      A     M    511.6;
      )     ;
      AN    M    519.2;
      AN    Q     30.4;
      =     Q     30.3;
NETWORK
TITLE =SLIDE BASE ADV LOCK'G REV

      A(    ;
      A     M    500.6;
      A     M    525.1;
      O     ;
      A     M    500.5;
      A     DB51.DBX    1.1;
      A     M    511.7;
      O     M    501.7;
      )     ;
      AN    M    519.3;
      AN    Q     30.3;
      =     Q     30.4;
NETWORK
TITLE =SLIDE BASE BREAK
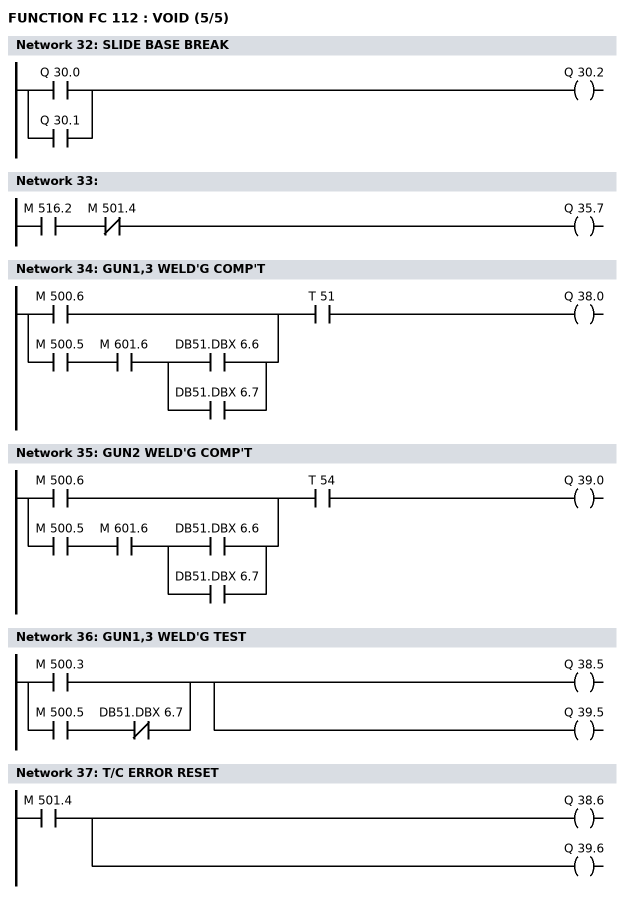

      O     Q     30.0;
      O     Q     30.1;
      =     Q     30.2;
NETWORK
TITLE =

      A     M    516.2;
      AN    M    501.4;
      =     Q     35.7;
NETWORK
TITLE =GUN1,3 WELD'G COMP'T

      A(    ;
      O     M    500.6;
      O     ;
      A     M    500.5;
      A     M    601.6;
      A(    ;
      O     DB51.DBX    6.6;
      O     DB51.DBX    6.7;
      )     ;
      )     ;
      A     T     51;
      =     Q     38.0;
NETWORK
TITLE =GUN2 WELD'G COMP'T

      A(    ;
      O     M    500.6;
      O     ;
      A     M    500.5;
      A     M    601.6;
      A(    ;
      O     DB51.DBX    6.6;
      O     DB51.DBX    6.7;
      )     ;
      )     ;
      A     T     54;
      =     Q     39.0;
NETWORK
TITLE =GUN1,3 WELD'G TEST

      O     M    500.3;
      O     ;
      A     M    500.5;
      AN    DB51.DBX    6.7;
      =     Q     38.5;
      =     Q     39.5;
NETWORK
TITLE =T/C ERROR RESET

      A     M    501.4;
      =     Q     38.6;
      =     Q     39.6;
NETWORK
TITLE =IDLE 공정

NETWORK
TITLE =

      AN    OV;
      =     L      0.0;
      A     L      0.0;
      A     I     32.0;
      AN    I     32.1;
      =     M    540.2;
      A     L      0.0;
      AN    I     32.0;
      A     I     32.1;
      =     M    540.3;
      A     L      0.0;
      A     I     33.0;
      AN    I     33.1;
      =     M    541.2;
      A     L      0.0;
      AN    I     33.0;
      A     I     33.1;
      =     M    541.3;
      A     L      0.0;
      A     I     33.2;
      AN    I     33.3;
      A     I     33.4;
      AN    I     33.5;
      =     M    541.4;
      A     L      0.0;
      AN    I     33.2;
      A     I     33.3;
      AN    I     33.4;
      A     I     33.5;
      =     M    541.5;
NETWORK
TITLE =
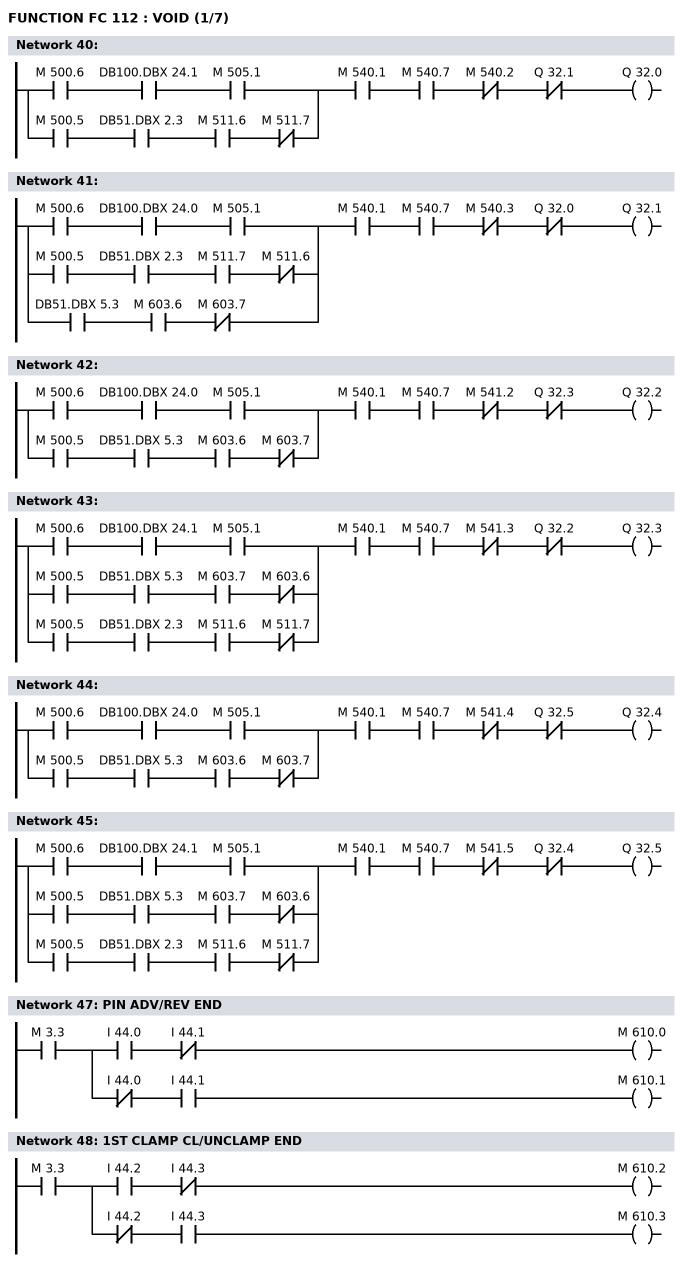

      A(    ;
      A     M    500.6;
      A     DB100.DBX   24.1;
      A     M    505.1;
      O     ;
      A     M    500.5;
      A     DB51.DBX    2.3;
      A     M    511.6;
      AN    M    511.7;
      )     ;
      A     M    540.1;
      A     M    540.7;
      AN    M    540.2;
      AN    Q     32.1;
      =     Q     32.0;
NETWORK
TITLE =

      A(    ;
      A     M    500.6;
      A     DB100.DBX   24.0;
      A     M    505.1;
      O     ;
      A     M    500.5;
      A     DB51.DBX    2.3;
      A     M    511.7;
      AN    M    511.6;
      O     ;
      A     DB51.DBX    5.3;
      A     M    603.6;
      AN    M    603.7;
      )     ;
      A     M    540.1;
      A     M    540.7;
      AN    M    540.3;
      AN    Q     32.0;
      =     Q     32.1;
NETWORK
TITLE =

      A(    ;
      A     M    500.6;
      A     DB100.DBX   24.0;
      A     M    505.1;
      O     ;
      A     M    500.5;
      A     DB51.DBX    5.3;
      A     M    603.6;
      AN    M    603.7;
      )     ;
      A     M    540.1;
      A     M    540.7;
      AN    M    541.2;
      AN    Q     32.3;
      =     Q     32.2;
NETWORK
TITLE =

      A(    ;
      A     M    500.6;
      A     DB100.DBX   24.1;
      A     M    505.1;
      O     ;
      A     M    500.5;
      A     DB51.DBX    5.3;
      A     M    603.7;
      AN    M    603.6;
      O     ;
      A     M    500.5;
      A     DB51.DBX    2.3;
      A     M    511.6;
      AN    M    511.7;
      )     ;
      A     M    540.1;
      A     M    540.7;
      AN    M    541.3;
      AN    Q     32.2;
      =     Q     32.3;
NETWORK
TITLE =

      A(    ;
      A     M    500.6;
      A     DB100.DBX   24.0;
      A     M    505.1;
      O     ;
      A     M    500.5;
      A     DB51.DBX    5.3;
      A     M    603.6;
      AN    M    603.7;
      )     ;
      A     M    540.1;
      A     M    540.7;
      AN    M    541.4;
      AN    Q     32.5;
      =     Q     32.4;
NETWORK
TITLE =

      A(    ;
      A     M    500.6;
      A     DB100.DBX   24.1;
      A     M    505.1;
      O     ;
      A     M    500.5;
      A     DB51.DBX    5.3;
      A     M    603.7;
      AN    M    603.6;
      O     ;
      A     M    500.5;
      A     DB51.DBX    2.3;
      A     M    511.6;
      AN    M    511.7;
      )     ;
      A     M    540.1;
      A     M    540.7;
      AN    M    541.5;
      AN    Q     32.4;
      =     Q     32.5;
NETWORK
TITLE =TL KEY 공정

NETWORK
TITLE =PIN ADV/REV END

      A     M      3.3;
      =     L      0.0;
      A     L      0.0;
      A     I     44.0;
      AN    I     44.1;
      =     M    610.0;
      A     L      0.0;
      AN    I     44.0;
      A     I     44.1;
      =     M    610.1;
NETWORK
TITLE =1ST CLAMP CL/UNCLAMP END

      A     M      3.3;
      =     L      0.0;
      A     L      0.0;
      A     I     44.2;
      AN    I     44.3;
      =     M    610.2;
      A     L      0.0;
      AN    I     44.2;
      A     I     44.3;
      =     M    610.3;
NETWORK
TITLE =2ND CLAMP CL/UNCLAMP END
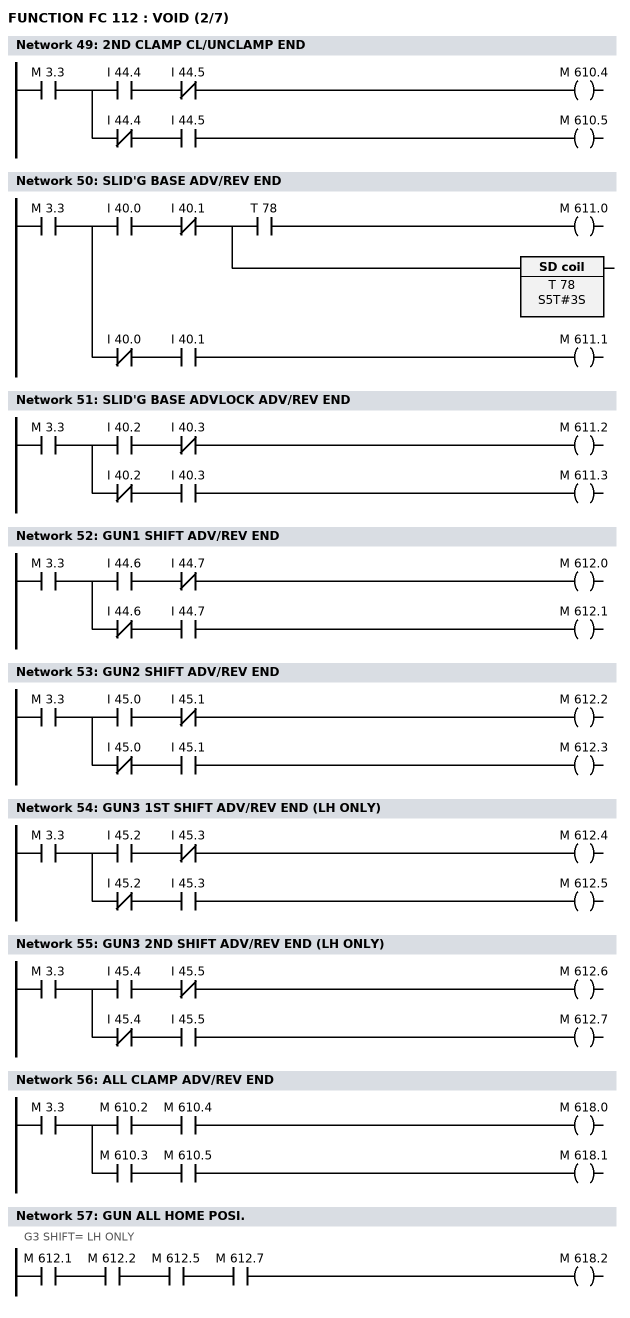

      A     M      3.3;
      =     L      0.0;
      A     L      0.0;
      A     I     44.4;
      AN    I     44.5;
      =     M    610.4;
      A     L      0.0;
      AN    I     44.4;
      A     I     44.5;
      =     M    610.5;
NETWORK
TITLE =SLID'G BASE ADV/REV END

      A     M      3.3;
      =     L      0.0;
      A     L      0.0;
      A     I     40.0;
      AN    I     40.1;
      =     L      0.1;
      A     L      0.1;
      A     T     78;
      =     M    611.0;
      A     L      0.1;
      BLD   102;
      L     S5T#3S;
      SD    T     78;
      A     L      0.0;
      AN    I     40.0;
      A     I     40.1;
      =     M    611.1;
NETWORK
TITLE =SLID'G BASE ADVLOCK ADV/REV END

      A     M      3.3;
      =     L      0.0;
      A     L      0.0;
      A     I     40.2;
      AN    I     40.3;
      =     M    611.2;
      A     L      0.0;
      AN    I     40.2;
      A     I     40.3;
      =     M    611.3;
NETWORK
TITLE =GUN1 SHIFT ADV/REV END

      A     M      3.3;
      =     L      0.0;
      A     L      0.0;
      A     I     44.6;
      AN    I     44.7;
      =     M    612.0;
      A     L      0.0;
      AN    I     44.6;
      A     I     44.7;
      =     M    612.1;
NETWORK
TITLE =GUN2 SHIFT ADV/REV END

